    |   movel(p[0.457444, -0.052609, -0.000100, 0.000000, -3.141593, 0.000000],accel_mss,speed_ms,0,0.000)
    |   movel(p[0.456698, -0.052972, -0.000100, 0.000000, -3.141593, 0.000000],accel_mss,speed_ms,0,0.000)
    |   movel(p[0.455801, -0.053375, -0.000100, 0.000000, -3.141593, 0.000000],accel_mss,speed_ms,0,0.000)
    |   movel(p[0.455556, -0.053469, -0.000100, 0.000000, -3.141593, 0.000000],accel_mss,speed_ms,0,0.000)
    |   movel(p[0.455254, -0.053564, -0.000100, 0.000000, 3.141593, 0.000000],accel_mss,speed_ms,0,0.000)
    |   movel(p[0.454943, -0.053645, -0.000100, 0.000000, -3.141593, 0.000000],accel_mss,speed_ms,0,0.000)
    |   movel(p[0.454676, -0.053699, -0.000100, 0.000000, -3.141593, 0.000000],accel_mss,speed_ms,0,0.000)
    |   movel(p[0.454424, -0.053742, -0.000100, 0.000000, -3.141593, 0.000000],accel_mss,speed_ms,0,0.000)
    |   movel(p[0.454164, -0.053792, -0.000100, 0.000000, -3.141593, 0.000000],accel_mss,speed_ms,0,0.000)
    |   movel(p[0.453931, -0.053841, -0.000100, 0.000000, -3.141593, 0.000000],accel_mss,speed_ms,0,0.000)
    |   movel(p[0.453776, -0.053881, -0.000100, 0.000000, -3.141593, 0.000000],accel_mss,speed_ms,0,0.000)
    |   movel(p[0.453611, -0.053919, -0.000100, 0.000000, 3.141593, 0.000000],accel_mss,speed_ms,0,0.000)
    |   movel(p[0.453619, -0.053815, -0.000100, 0.000000, 3.141593, 0.000000],accel_mss,speed_ms,0,0.000)
    |   movel(p[0.453839, -0.053573, -0.000100, 0.000000, -3.141593, 0.000000],accel_mss,speed_ms,0,0.000)
    |   movel(p[0.453990, -0.053422, -0.000100, 0.000000, -3.141593, 0.000000],accel_mss,speed_ms,0,0.000)
    |   movel(p[0.454143, -0.053294, -0.000100, 0.000000, -3.141593, 0.000000],accel_mss,speed_ms,0,0.000)
    |   movel(p[0.454280, -0.053201, -0.000100, 0.000000, -3.141593, 0.000000],accel_mss,speed_ms,0,0.000)
    |   movel(p[0.454467, -0.053141, -0.000100, 0.000000, -3.141593, 0.000000],accel_mss,speed_ms,0,0.000)
    |   movel(p[0.454831, -0.052851, -0.000100, 0.000000, -3.141593, 0.000000],accel_mss,speed_ms,0,0.000)
    |   movel(p[0.455254, -0.052494, -0.000100, 0.000000, -3.141593, 0.000000],accel_mss,speed_ms,0,0.000)
    |   movel(p[0.455726, -0.052070, -0.000100, 0.000000, -3.141593, 0.000000],accel_mss,speed_ms,0,0.000)
    |   movel(p[0.456326, -0.051518, -0.000100, 0.000000, -3.141593, 0.000000],accel_mss,speed_ms,0,0.000)
    |   movel(p[0.456926, -0.050965, -0.000100, 0.000000, -3.141593, 0.000000],accel_mss,speed_ms,0,0.000)
    |   movel(p[0.456738, -0.050804, -0.000100, 0.000000, -3.141593, 0.000000],accel_mss,speed_ms,0,0.000)
    |   movel(p[0.456551, -0.050642, -0.000100, 0.000000, -3.141593, 0.000000],accel_mss,speed_ms,0,0.000)
    |   movel(p[0.456382, -0.050508, -0.000100, 0.000000, -3.141593, 0.000000],accel_mss,speed_ms,0,0.000)
    |   movel(p[0.456187, -0.050372, -0.000100, 0.000000, -3.141593, 0.000000],accel_mss,speed_ms,0,0.000)
    |   movel(p[0.455994, -0.050254, -0.000100, 0.000000, -3.141593, 0.000000],accel_mss,speed_ms,0,0.000)
    |   movel(p[0.455838, -0.050177, -0.000100, 0.000000, 3.141593, 0.000000],accel_mss,speed_ms,0,0.000)
    |   movel(p[0.455624, -0.049995, -0.000100, 0.000000, 3.141593, 0.000000],accel_mss,speed_ms,0,0.000)
    |   movel(p[0.455507, -0.049685, -0.000100, 0.000000, -3.141593, 0.000000],accel_mss,speed_ms,0,0.000)
    |   movel(p[0.455509, -0.049322, -0.000100, 0.000000, -3.141593, 0.000000],accel_mss,speed_ms,0,0.000)
    |   movel(p[0.455638, -0.048995, -0.000100, 0.000000, -3.141593, 0.000000],accel_mss,speed_ms,0,0.000)
    |   movel(p[0.455763, -0.048888, -0.000100, 0.000000, 3.141593, 0.000000],accel_mss,speed_ms,0,0.000)
    |   movel(p[0.455918, -0.048877, -0.000100, 0.000000, 3.141593, 0.000000],accel_mss,speed_ms,0,0.000)
    |   movel(p[0.456158, -0.048983, -0.000100, 0.000000, -3.141593, 0.000000],accel_mss,speed_ms,0,0.000)
    |   movel(p[0.456626, -0.049278, -0.000100, 0.000000, 3.141593, 0.000000],accel_mss,speed_ms,0,0.000)
    |   movel(p[0.456820, -0.049403, -0.000100, 0.000000, -3.141593, 0.000000],accel_mss,speed_ms,0,0.000)
    |   movel(p[0.457032, -0.049532, -0.000100, 0.000000, -3.141593, 0.000000],accel_mss,speed_ms,0,0.000)
    |   movel(p[0.457229, -0.049648, -0.000100, 0.000000, -3.141593, 0.000000],accel_mss,speed_ms,0,0.000)
    |   movel(p[0.457376, -0.049726, -0.000100, 0.000000, -3.141593, 0.000000],accel_mss,speed_ms,0,0.000)
    |   movel(p[0.457509, -0.049798, -0.000100, 0.000000, -3.141593, 0.000000],accel_mss,speed_ms,0,0.000)
    |   movel(p[0.457663, -0.049888, -0.000100, 0.000000, -3.141593, 0.000000],accel_mss,speed_ms,0,0.000)
    |   movel(p[0.457813, -0.049981, -0.000100, 0.000000, -3.141593, 0.000000],accel_mss,speed_ms,0,0.000)
    |   movel(p[0.457933, -0.050062, -0.000100, 0.000000, 3.141593, 0.000000],accel_mss,speed_ms,0,0.000)
    |   movel(p[0.458085, -0.050138, -0.000100, 0.000000, 3.141593, 0.000000],accel_mss,speed_ms,0,0.000)
    |   movel(p[0.458220, -0.050138, -0.000100, 0.000000, -3.141593, 0.000000],accel_mss,speed_ms,0,0.000)
    |   movel(p[0.458374, -0.050057, -0.000100, 0.000000, -3.141593, 0.000000],accel_mss,speed_ms,0,0.000)
    |   movel(p[0.458608, -0.049856, -0.000100, 0.000000, -3.141593, 0.000000],accel_mss,speed_ms,0,0.000)
    |   movel(p[0.458781, -0.049703, -0.000100, 0.000000, -3.141593, 0.000000],accel_mss,speed_ms,0,0.000)
    |   movel(p[0.458954, -0.049564, -0.000100, 0.000000, -3.141593, 0.000000],accel_mss,speed_ms,0,0.000)
    |   movel(p[0.459108, -0.049455, -0.000100, 0.000000, -3.141593, 0.000000],accel_mss,speed_ms,0,0.000)
    |   movel(p[0.459201, -0.049410, -0.000100, 0.000000, -3.141593, 0.000000],accel_mss,speed_ms,0,0.000)
    |   movel(p[0.459315, -0.049350, -0.000100, 0.000000, -3.141593, 0.000000],accel_mss,speed_ms,0,0.000)
    |   movel(p[0.459714, -0.049032, -0.000100, 0.000000, 3.141593, 0.000000],accel_mss,speed_ms,0,0.000)
    |   movel(p[0.460181, -0.048647, -0.000100, 0.000000, -3.141593, 0.000000],accel_mss,speed_ms,0,0.000)
    |   movel(p[0.460701, -0.048201, -0.000100, 0.000000, -3.141593, 0.000000],accel_mss,speed_ms,0,0.000)
    |   movel(p[0.462085, -0.046990, -0.000100, 0.000000, -3.141593, 0.000000],accel_mss,speed_ms,0,0.001)
    |   movel(p[0.462714, -0.046416, -0.000100, 0.000000, -3.141593, 0.000000],accel_mss,speed_ms,0,0.000)
    |   movel(p[0.463064, -0.046063, -0.000100, 0.000000, -3.141593, 0.000000],accel_mss,speed_ms,0,0.000)
    |   movel(p[0.463140, -0.045885, -0.000100, 0.000000, -3.141593, 0.000000],accel_mss,speed_ms,0,0.000)
    |   movel(p[0.463215, -0.045710, -0.000100, 0.000000, -3.141593, 0.000000],accel_mss,speed_ms,0,0.000)
    |   movel(p[0.463291, -0.045611, -0.000100, 0.000000, 3.141593, 0.000000],accel_mss,speed_ms,0,0.000)
    |   movel(p[0.463379, -0.045526, -0.000100, 0.000000, -3.141593, 0.000000],accel_mss,speed_ms,0,0.000)
    |   movel(p[0.463505, -0.045328, -0.000100, 0.000000, -3.141593, 0.000000],accel_mss,speed_ms,0,0.000)
    |   movel(p[0.463516, -0.045062, -0.000100, 0.000000, -3.141593, 0.000000],accel_mss,speed_ms,0,0.000)
    |   movel(p[0.463406, -0.044754, -0.000100, 0.000000, -3.141593, 0.000000],accel_mss,speed_ms,0,0.000)
    |   movel(p[0.463185, -0.044441, -0.000100, 0.000000, -3.141593, 0.000000],accel_mss,speed_ms,0,0.000)
    |   movel(p[0.462587, -0.044166, -0.000100, 0.000000, -3.141593, 0.000000],accel_mss,speed_ms,0,0.000)
    |   movel(p[0.461450, -0.044260, -0.000100, 0.000000, -3.141593, 0.000000],accel_mss,speed_ms,0,0.000)
    |   movel(p[0.460266, -0.044596, -0.000100, 0.000000, -3.141593, 0.000000],accel_mss,speed_ms,0,0.000)
    |   movel(p[0.459446, -0.045117, -0.000100, 0.000000, -3.141593, 0.000000],accel_mss,speed_ms,0,0.000)
    |   movel(p[0.459259, -0.045315, -0.000100, 0.000000, 3.141593, 0.000000],accel_mss,speed_ms,0,0.000)
    |   movel(p[0.459093, -0.045532, -0.000100, 0.000000, -3.141593, 0.000000],accel_mss,speed_ms,0,0.000)
    |   movel(p[0.458970, -0.045736, -0.000100, 0.000000, -3.141593, 0.000000],accel_mss,speed_ms,0,0.000)
    |   movel(p[0.458921, -0.045889, -0.000100, 0.000000, -3.141593, 0.000000],accel_mss,speed_ms,0,0.000)
    |   movel(p[0.458835, -0.046155, -0.000100, 0.000000, -3.141593, 0.000000],accel_mss,speed_ms,0,0.000)
    |   movel(p[0.458710, -0.046179, -0.000100, 0.000000, -3.141593, 0.000000],accel_mss,speed_ms,0,0.000)
    |   movel(p[0.458578, -0.045966, -0.000100, 0.000000, -3.141593, 0.000000],accel_mss,speed_ms,0,0.000)
    |   movel(p[0.458501, -0.045529, -0.000100, 0.000000, -3.141593, 0.000000],accel_mss,speed_ms,0,0.000)
    |   movel(p[0.458463, -0.045191, -0.000100, 0.000000, 3.141593, 0.000000],accel_mss,speed_ms,0,0.000)
    |   movel(p[0.458426, -0.044854, -0.000100, 0.000000, -3.141593, 0.000000],accel_mss,speed_ms,0,0.000)
    |   movel(p[0.457956, -0.044809, -0.000100, 0.000000, -3.141593, 0.000000],accel_mss,speed_ms,0,0.000)
    |   movel(p[0.457486, -0.044764, -0.000100, 0.000000, -3.141593, 0.000000],accel_mss,speed_ms,0,0.000)
    |   movel(p[0.457118, -0.044722, -0.000100, 0.000000, -3.141593, 0.000000],accel_mss,speed_ms,0,0.000)
    |   movel(p[0.456793, -0.044671, -0.000100, 0.000000, -3.141593, 0.000000],accel_mss,speed_ms,0,0.000)
    |   movel(p[0.456525, -0.044617, -0.000100, 0.000000, -3.141593, 0.000000],accel_mss,speed_ms,0,0.000)
    |   movel(p[0.456394, -0.044568, -0.000100, 0.000000, -3.141593, 0.000000],accel_mss,speed_ms,0,0.000)
    |   movel(p[0.456241, -0.044747, -0.000100, 0.000000, -3.141593, 0.000000],accel_mss,speed_ms,0,0.000)
    |   movel(p[0.456164, -0.044906, -0.000100, 0.000000, -3.141593, 0.000000],accel_mss,speed_ms,0,0.000)
    |   movel(p[0.456062, -0.045092, -0.000100, 0.000000, -3.141593, 0.000000],accel_mss,speed_ms,0,0.000)
    |   movel(p[0.455929, -0.045243, -0.000100, 0.000000, 3.141593, 0.000000],accel_mss,speed_ms,0,0.000)
    |   movel(p[0.455772, -0.045351, -0.000100, 0.000000, -3.141593, 0.000000],accel_mss,speed_ms,0,0.000)
    |   movel(p[0.455599, -0.045411, -0.000100, 0.000000, -3.141593, 0.000000],accel_mss,speed_ms,0,0.000)
    |   movel(p[0.455393, -0.045435, -0.000100, 0.000000, -3.141593, 0.000000],accel_mss,speed_ms,0,0.000)
    |   movel(p[0.455279, -0.045400, -0.000100, 0.000000, -3.141593, 0.000000],accel_mss,speed_ms,0,0.000)
    |   movel(p[0.455211, -0.045303, -0.000100, 0.000000, -3.141593, 0.000000],accel_mss,speed_ms,0,0.000)
    |   movel(p[0.455171, -0.045103, -0.000100, 0.000000, -3.141593, 0.000000],accel_mss,speed_ms,0,0.000)
    |   movel(p[0.454942, -0.044704, -0.000100, 0.000000, -3.141593, 0.000000],accel_mss,speed_ms,0,0.000)
    |   movel(p[0.454225, -0.044245, -0.000100, 0.000000, -3.141593, 0.000000],accel_mss,speed_ms,0,0.000)
    |   movel(p[0.453175, -0.043770, -0.000100, 0.000000, -3.141593, 0.000000],accel_mss,speed_ms,0,0.000)
    |   movel(p[0.451809, -0.043308, -0.000100, 0.000000, -3.141593, 0.000000],accel_mss,speed_ms,0,0.001)
    |   movel(p[0.450322, -0.042878, -0.000100, 0.000000, 3.141593, 0.000000],accel_mss,speed_ms,0,0.001)
    |   movel(p[0.449341, -0.042643, -0.000100, 0.000000, -3.141593, 0.000000],accel_mss,speed_ms,0,0.000)
    |   movel(p[0.448468, -0.042508, -0.000100, 0.000000, -3.141593, 0.000000],accel_mss,speed_ms,0,0.000)
    |   movel(p[0.447398, -0.042420, -0.000100, 0.000000, -3.141593, 0.000000],accel_mss,speed_ms,0,0.000)
    |   movel(p[0.445629, -0.042470, -0.000100, 0.000000, -3.141593, 0.000000],accel_mss,speed_ms,0,0.001)
    |   movel(p[0.444085, -0.042832, -0.000100, 0.000000, -3.141593, 0.000000],accel_mss,speed_ms,0,0.001)
    |   movel(p[0.442690, -0.043537, -0.000100, 0.000000, -3.141593, 0.000000],accel_mss,speed_ms,0,0.001)
    |   movel(p[0.441363, -0.044610, -0.000100, 0.000000, -3.141593, 0.000000],accel_mss,speed_ms,0,0.001)
    |   movel(p[0.440975, -0.045000, -0.000100, 0.000000, -3.141593, 0.000000],accel_mss,speed_ms,0,0.000)
    |   movel(p[0.440648, -0.045357, -0.000100, 0.000000, -3.141593, 0.000000],accel_mss,speed_ms,0,0.000)
    |   movel(p[0.440388, -0.045663, -0.000100, 0.000000, -3.141593, 0.000000],accel_mss,speed_ms,0,0.000)
    |   movel(p[0.440351, -0.045769, -0.000100, 0.000000, -3.141593, 0.000000],accel_mss,speed_ms,0,0.000)
    |   movel(p[0.440286, -0.045945, -0.000100, 0.000000, 3.141593, 0.000000],accel_mss,speed_ms,0,0.000)
    |   movel(p[0.440214, -0.046043, -0.000100, 0.000000, -3.141593, 0.000000],accel_mss,speed_ms,0,0.000)
    |   movel(p[0.440129, -0.046126, -0.000100, 0.000000, -3.141593, 0.000000],accel_mss,speed_ms,0,0.000)
    |   movel(p[0.439825, -0.046492, -0.000100, 0.000000, -3.141593, 0.000000],accel_mss,speed_ms,0,0.000)
    |   movel(p[0.439490, -0.047169, -0.000100, 0.000000, -3.141593, 0.000000],accel_mss,speed_ms,0,0.000)
    |   movel(p[0.439225, -0.047864, -0.000100, 0.000000, -3.141593, 0.000000],accel_mss,speed_ms,0,0.000)
    |   movel(p[0.439223, -0.048220, -0.000100, 0.000000, -3.141593, 0.000000],accel_mss,speed_ms,0,0.000)
    |   movel(p[0.439220, -0.048445, -0.000100, 0.000000, -3.141593, 0.000000],accel_mss,speed_ms,0,0.000)
    |   movel(p[0.439086, -0.048517, -0.000100, 0.000000, -3.141593, 0.000000],accel_mss,speed_ms,0,0.000)
    |   movel(p[0.438794, -0.048368, -0.000100, 0.000000, -3.141593, 0.000000],accel_mss,speed_ms,0,0.000)
    |   movel(p[0.438401, -0.048004, -0.000100, 0.000000, -3.141593, 0.000000],accel_mss,speed_ms,0,0.000)
    |   movel(p[0.438193, -0.047803, -0.000100, 0.000000, -3.141593, 0.000000],accel_mss,speed_ms,0,0.000)
    |   movel(p[0.437991, -0.047633, -0.000100, 0.000000, -3.141593, 0.000000],accel_mss,speed_ms,0,0.000)
    |   movel(p[0.437816, -0.047507, -0.000100, 0.000000, 3.141593, 0.000000],accel_mss,speed_ms,0,0.000)
    |   movel(p[0.437634, -0.047455, -0.000100, 0.000000, -3.141593, 0.000000],accel_mss,speed_ms,0,0.000)
    |   movel(p[0.437496, -0.047365, -0.000100, 0.000000, 3.141593, 0.000000],accel_mss,speed_ms,0,0.000)
    |   movel(p[0.437341, -0.047239, -0.000100, 0.000000, -3.141593, 0.000000],accel_mss,speed_ms,0,0.000)
    |   movel(p[0.437189, -0.047090, -0.000100, 0.000000, -3.141593, 0.000000],accel_mss,speed_ms,0,0.000)
    |   movel(p[0.436313, -0.046354, -0.000100, 0.000000, -3.141593, 0.000000],accel_mss,speed_ms,0,0.000)
    |   movel(p[0.434998, -0.045590, -0.000100, 0.000000, 3.141593, 0.000000],accel_mss,speed_ms,0,0.001)
    |   movel(p[0.433551, -0.044941, -0.000100, 0.000000, -3.141593, 0.000000],accel_mss,speed_ms,0,0.001)
    |   movel(p[0.432241, -0.044552, -0.000100, 0.000000, -3.141593, 0.000000],accel_mss,speed_ms,0,0.001)
    |   movel(p[0.431305, -0.044404, -0.000100, 0.000000, -3.141593, 0.000000],accel_mss,speed_ms,0,0.000)
    |   movel(p[0.430304, -0.044342, -0.000100, 0.000000, -3.141593, 0.000000],accel_mss,speed_ms,0,0.000)
    |   movel(p[0.429265, -0.044365, -0.000100, 0.000000, 3.141593, 0.000000],accel_mss,speed_ms,0,0.000)
    |   movel(p[0.428220, -0.044473, -0.000100, 0.000000, -3.141593, 0.000000],accel_mss,speed_ms,0,0.000)
    |   movel(p[0.427528, -0.044623, -0.000100, 0.000000, 3.141593, 0.000000],accel_mss,speed_ms,0,0.000)
    |   movel(p[0.426799, -0.044878, -0.000100, 0.000000, -3.141593, 0.000000],accel_mss,speed_ms,0,0.000)
    |   movel(p[0.426044, -0.045234, -0.000100, 0.000000, -3.141593, 0.000000],accel_mss,speed_ms,0,0.000)
    |   movel(p[0.425276, -0.045686, -0.000100, 0.000000, -3.141593, 0.000000],accel_mss,speed_ms,0,0.000)
    |   movel(p[0.425087, -0.045804, -0.000100, 0.000000, -3.141593, 0.000000],accel_mss,speed_ms,0,0.000)
    |   movel(p[0.424892, -0.045920, -0.000100, 0.000000, 3.141593, 0.000000],accel_mss,speed_ms,0,0.000)
    |   movel(p[0.424717, -0.046019, -0.000100, 0.000000, 3.141593, 0.000000],accel_mss,speed_ms,0,0.000)
    |   movel(p[0.424601, -0.046077, -0.000100, 0.000000, -3.141593, 0.000000],accel_mss,speed_ms,0,0.000)
    |   movel(p[0.424480, -0.046142, -0.000100, 0.000000, -3.141593, 0.000000],accel_mss,speed_ms,0,0.000)
    |   movel(p[0.424281, -0.046274, -0.000100, 0.000000, -3.141593, 0.000000],accel_mss,speed_ms,0,0.000)
    |   movel(p[0.424055, -0.046434, -0.000100, 0.000000, 3.141593, 0.000000],accel_mss,speed_ms,0,0.000)
    |   movel(p[0.423829, -0.046604, -0.000100, 0.000000, -3.141593, 0.000000],accel_mss,speed_ms,0,0.000)
    |   movel(p[0.423610, -0.046767, -0.000100, 0.000000, -3.141593, 0.000000],accel_mss,speed_ms,0,0.000)
    |   movel(p[0.423402, -0.046904, -0.000100, 0.000000, 3.141593, 0.000000],accel_mss,speed_ms,0,0.000)
    |   movel(p[0.423225, -0.047008, -0.000100, 0.000000, 3.141593, 0.000000],accel_mss,speed_ms,0,0.000)
    |   movel(p[0.422935, -0.047109, -0.000100, 0.000000, -3.141593, 0.000000],accel_mss,speed_ms,0,0.000)
    |   movel(p[0.422672, -0.047388, -0.000100, 0.000000, 3.141593, 0.000000],accel_mss,speed_ms,0,0.000)
    |   movel(p[0.422465, -0.047699, -0.000100, 0.000000, -3.141593, 0.000000],accel_mss,speed_ms,0,0.000)
    |   movel(p[0.422470, -0.047879, -0.000100, 0.000000, -3.141593, 0.000000],accel_mss,speed_ms,0,0.000)
    |   movel(p[0.422558, -0.047959, -0.000100, 0.000000, -3.141593, 0.000000],accel_mss,speed_ms,0,0.000)
    |   movel(p[0.422809, -0.048074, -0.000100, 0.000000, 3.141593, 0.000000],accel_mss,speed_ms,0,0.000)
    |   movel(p[0.423123, -0.048195, -0.000100, 0.000000, -3.141593, 0.000000],accel_mss,speed_ms,0,0.000)
    |   movel(p[0.423476, -0.048306, -0.000100, 0.000000, 3.141593, 0.000000],accel_mss,speed_ms,0,0.000)
    |   movel(p[0.423831, -0.048414, -0.000100, 0.000000, -3.141593, 0.000000],accel_mss,speed_ms,0,0.000)
    |   movel(p[0.424153, -0.048526, -0.000100, 0.000000, -3.141593, 0.000000],accel_mss,speed_ms,0,0.000)
    |   movel(p[0.424417, -0.048630, -0.000100, 0.000000, -3.141593, 0.000000],accel_mss,speed_ms,0,0.000)
    |   movel(p[0.424518, -0.048696, -0.000100, 0.000000, -3.141593, 0.000000],accel_mss,speed_ms,0,0.000)
    |   movel(p[0.424691, -0.048790, -0.000100, 0.000000, -3.141593, 0.000000],accel_mss,speed_ms,0,0.000)
    |   movel(p[0.424803, -0.048819, -0.000100, 0.000000, -3.141593, 0.000000],accel_mss,speed_ms,0,0.000)
    |   movel(p[0.424908, -0.048829, -0.000100, 0.000000, -3.141593, 0.000000],accel_mss,speed_ms,0,0.000)
    |   movel(p[0.425036, -0.048845, -0.000100, 0.000000, -3.141593, 0.000000],accel_mss,speed_ms,0,0.000)
    |   movel(p[0.425230, -0.048903, -0.000100, 0.000000, 3.141593, 0.000000],accel_mss,speed_ms,0,0.000)
    |   movel(p[0.425448, -0.048984, -0.000100, 0.000000, -3.141593, 0.000000],accel_mss,speed_ms,0,0.000)
    |   movel(p[0.425659, -0.049081, -0.000100, 0.000000, -3.141593, 0.000000],accel_mss,speed_ms,0,0.000)
    |   movel(p[0.425911, -0.049179, -0.000100, 0.000000, -3.141593, 0.000000],accel_mss,speed_ms,0,0.000)
    |   movel(p[0.426235, -0.049257, -0.000100, 0.000000, -3.141593, 0.000000],accel_mss,speed_ms,0,0.000)
    |   movel(p[0.426586, -0.049306, -0.000100, 0.000000, -3.141593, 0.000000],accel_mss,speed_ms,0,0.000)
    |   movel(p[0.426920, -0.049319, -0.000100, 0.000000, -3.141593, 0.000000],accel_mss,speed_ms,0,0.000)
    |   movel(p[0.427388, -0.049310, -0.000100, 0.000000, -3.141593, 0.000000],accel_mss,speed_ms,0,0.000)
    |   movel(p[0.428446, -0.049289, -0.000100, 0.000000, 3.141593, 0.000000],accel_mss,speed_ms,0,0.000)
    |   movel(p[0.429706, -0.049264, -0.000100, 0.000000, -3.141593, 0.000000],accel_mss,speed_ms,0,0.001)
    |   movel(p[0.431055, -0.049237, -0.000100, 0.000000, -3.141593, 0.000000],accel_mss,speed_ms,0,0.001)
    |   movel(p[0.433370, -0.049228, -0.000100, 0.000000, -3.141593, 0.000000],accel_mss,speed_ms,0,0.001)
    |   movel(p[0.435193, -0.049311, -0.000100, 0.000000, -3.141593, 0.000000],accel_mss,speed_ms,0,0.001)
    |   movel(p[0.436687, -0.049489, -0.000100, 0.000000, -3.141593, 0.000000],accel_mss,speed_ms,0,0.001)
    |   movel(p[0.437970, -0.049777, -0.000100, 0.000000, -3.141593, 0.000000],accel_mss,speed_ms,0,0.001)
    |   movel(p[0.438501, -0.049999, -0.000100, 0.000000, -3.141593, 0.000000],accel_mss,speed_ms,0,0.000)
    |   movel(p[0.438479, -0.050152, -0.000100, 0.000000, -3.141593, 0.000000],accel_mss,speed_ms,0,0.000)
    |   movel(p[0.437782, -0.050237, -0.000100, 0.000000, -3.141593, 0.000000],accel_mss,speed_ms,0,0.000)
    |   movel(p[0.435923, -0.050249, -0.000100, 0.000000, 3.141593, 0.000000],accel_mss,speed_ms,0,0.001)
    |   movel(p[0.433512, -0.050292, -0.000100, 0.000000, 3.141593, 0.000000],accel_mss,speed_ms,0,0.001)
    |   movel(p[0.431714, -0.050442, -0.000100, 0.000000, -3.141593, 0.000000],accel_mss,speed_ms,0,0.001)
    |   movel(p[0.430039, -0.050745, -0.000100, 0.000000, -3.141593, 0.000000],accel_mss,speed_ms,0,0.001)
    |   movel(p[0.428051, -0.051269, -0.000100, 0.000000, -3.141593, 0.000000],accel_mss,speed_ms,0,0.001)
    |   movel(p[0.427120, -0.051615, -0.000100, 0.000000, -3.141593, 0.000000],accel_mss,speed_ms,0,0.000)
    |   movel(p[0.425780, -0.052258, -0.000100, 0.000000, -3.141593, 0.000000],accel_mss,speed_ms,0,0.001)
    |   movel(p[0.424487, -0.052945, -0.000100, 0.000000, -3.141593, 0.000000],accel_mss,speed_ms,0,0.001)
    |   movel(p[0.423864, -0.053391, -0.000100, 0.000000, -3.141593, 0.000000],accel_mss,speed_ms,0,0.000)
    |   movel(p[0.423754, -0.053482, -0.000100, 0.000000, -3.141593, 0.000000],accel_mss,speed_ms,0,0.000)
    |   movel(p[0.423639, -0.053559, -0.000100, 0.000000, -3.141593, 0.000000],accel_mss,speed_ms,0,0.000)
    |   movel(p[0.423535, -0.053614, -0.000100, 0.000000, -3.141593, 0.000000],accel_mss,speed_ms,0,0.000)
    |   movel(p[0.423234, -0.053725, -0.000100, 0.000000, -3.141593, 0.000000],accel_mss,speed_ms,0,0.000)
    |   movel(p[0.421486, -0.055471, -0.000100, 0.000000, -3.141593, 0.000000],accel_mss,speed_ms,0,0.001)
    |   movel(p[0.419747, -0.057225, -0.000100, 0.000000, -3.141593, 0.000000],accel_mss,speed_ms,0,0.001)
    |   movel(p[0.419651, -0.057459, -0.000100, 0.000000, -3.141593, 0.000000],accel_mss,speed_ms,0,0.000)
    |   movel(p[0.419474, -0.057743, -0.000100, 0.000000, 3.141593, 0.000000],accel_mss,speed_ms,0,0.000)
    |   movel(p[0.419280, -0.057968, -0.000100, 0.000000, -3.141593, 0.000000],accel_mss,speed_ms,0,0.000)
    |   movel(p[0.419051, -0.058204, -0.000100, 0.000000, -3.141593, 0.000000],accel_mss,speed_ms,0,0.000)
    |   movel(p[0.418821, -0.058440, -0.000100, 0.000000, -3.141593, 0.000000],accel_mss,speed_ms,0,0.000)
    |   movel(p[0.418627, -0.058665, -0.000100, 0.000000, 3.141593, 0.000000],accel_mss,speed_ms,0,0.000)
    |   movel(p[0.418480, -0.058860, -0.000100, 0.000000, -3.141593, 0.000000],accel_mss,speed_ms,0,0.000)
    |   movel(p[0.418418, -0.059049, -0.000100, 0.000000, -3.141593, 0.000000],accel_mss,speed_ms,0,0.000)
    |   movel(p[0.418230, -0.059284, -0.000100, 0.000000, -3.141593, 0.000000],accel_mss,speed_ms,0,0.000)
    |   movel(p[0.417988, -0.059559, -0.000100, 0.000000, -3.141593, 0.000000],accel_mss,speed_ms,0,0.000)
    |   movel(p[0.417701, -0.059854, -0.000100, 0.000000, -3.141593, 0.000000],accel_mss,speed_ms,0,0.000)
    |   movel(p[0.417413, -0.060146, -0.000100, 0.000000, -3.141593, 0.000000],accel_mss,speed_ms,0,0.000)
    |   movel(p[0.417171, -0.060410, -0.000100, 0.000000, -3.141593, 0.000000],accel_mss,speed_ms,0,0.000)
    |   movel(p[0.416977, -0.060638, -0.000100, 0.000000, -3.141593, 0.000000],accel_mss,speed_ms,0,0.000)
    |   movel(p[0.416978, -0.060756, -0.000100, 0.000000, -3.141593, 0.000000],accel_mss,speed_ms,0,0.000)
    |   movel(p[0.417072, -0.060794, -0.000100, 0.000000, -3.141593, 0.000000],accel_mss,speed_ms,0,0.000)
    |   movel(p[0.417205, -0.060821, -0.000100, 0.000000, 3.141593, 0.000000],accel_mss,speed_ms,0,0.000)
    |   movel(p[0.417363, -0.060830, -0.000100, 0.000000, -3.141593, 0.000000],accel_mss,speed_ms,0,0.000)
    |   movel(p[0.417987, -0.060788, -0.000100, 0.000000, -3.141593, 0.000000],accel_mss,speed_ms,0,0.000)
    |   movel(p[0.419857, -0.060521, -0.000100, 0.000000, -3.141593, 0.000000],accel_mss,speed_ms,0,0.001)
    |   movel(p[0.421692, -0.060242, -0.000100, 0.000000, -3.141593, 0.000000],accel_mss,speed_ms,0,0.001)
    |   movel(p[0.422501, -0.060076, -0.000100, 0.000000, -3.141593, 0.000000],accel_mss,speed_ms,0,0.000)
    |   movel(p[0.422801, -0.060010, -0.000100, 0.000000, -3.141593, 0.000000],accel_mss,speed_ms,0,0.000)
    |   movel(p[0.423353, -0.059908, -0.000100, 0.000000, -3.141593, 0.000000],accel_mss,speed_ms,0,0.000)
    |   movel(p[0.423999, -0.059798, -0.000100, 0.000000, -3.141593, 0.000000],accel_mss,speed_ms,0,0.000)
    |   movel(p[0.424665, -0.059692, -0.000100, 0.000000, -3.141593, 0.000000],accel_mss,speed_ms,0,0.000)
    |   movel(p[0.426937, -0.059271, -0.000100, 0.000000, 3.141593, 0.000000],accel_mss,speed_ms,0,0.001)
    |   movel(p[0.429210, -0.058707, -0.000100, 0.000000, -3.141593, 0.000000],accel_mss,speed_ms,0,0.001)
    |   movel(p[0.431205, -0.058082, -0.000100, 0.000000, -3.141593, 0.000000],accel_mss,speed_ms,0,0.001)
    |   movel(p[0.432551, -0.057484, -0.000100, 0.000000, -3.141593, 0.000000],accel_mss,speed_ms,0,0.001)
    |   movel(p[0.432888, -0.057299, -0.000100, 0.000000, -3.141593, 0.000000],accel_mss,speed_ms,0,0.000)
    |   movel(p[0.433221, -0.057117, -0.000100, 0.000000, -3.141593, 0.000000],accel_mss,speed_ms,0,0.000)
    |   movel(p[0.433509, -0.056959, -0.000100, 0.000000, -3.141593, 0.000000],accel_mss,speed_ms,0,0.000)
    |   movel(p[0.433676, -0.056868, -0.000100, 0.000000, -3.141593, 0.000000],accel_mss,speed_ms,0,0.000)
    |   movel(p[0.434155, -0.056529, -0.000100, 0.000000, 3.141593, 0.000000],accel_mss,speed_ms,0,0.000)
    |   movel(p[0.434933, -0.055797, -0.000100, 0.000000, -3.141593, 0.000000],accel_mss,speed_ms,0,0.000)
    |   movel(p[0.435685, -0.055018, -0.000100, 0.000000, -3.141593, 0.000000],accel_mss,speed_ms,0,0.000)
    |   movel(p[0.436125, -0.054454, -0.000100, 0.000000, -3.141593, 0.000000],accel_mss,speed_ms,0,0.000)
    |   movel(p[0.436484, -0.053902, -0.000100, 0.000000, -3.141593, 0.000000],accel_mss,speed_ms,0,0.000)
    |   movel(p[0.436721, -0.053523, -0.000100, 0.000000, -3.141593, 0.000000],accel_mss,speed_ms,0,0.000)
    |   movel(p[0.436891, -0.053227, -0.000100, 0.000000, -3.141593, 0.000000],accel_mss,speed_ms,0,0.000)
    |   movel(p[0.437030, -0.052954, -0.000100, 0.000000, -3.141593, 0.000000],accel_mss,speed_ms,0,0.000)
    |   movel(p[0.437118, -0.052806, -0.000100, 0.000000, -3.141593, 0.000000],accel_mss,speed_ms,0,0.000)
    |   movel(p[0.437281, -0.052597, -0.000100, 0.000000, -3.141593, 0.000000],accel_mss,speed_ms,0,0.000)
    |   movel(p[0.437480, -0.052371, -0.000100, 0.000000, -3.141593, 0.000000],accel_mss,speed_ms,0,0.000)
    |   movel(p[0.437687, -0.052160, -0.000100, 0.000000, 3.141593, 0.000000],accel_mss,speed_ms,0,0.000)
    |   movel(p[0.438114, -0.051835, -0.000100, 0.000000, -3.141593, 0.000000],accel_mss,speed_ms,0,0.000)
    |   movel(p[0.438368, -0.051872, -0.000100, 0.000000, -3.141593, 0.000000],accel_mss,speed_ms,0,0.000)
    |   movel(p[0.438519, -0.052214, -0.000100, 0.000000, -3.141593, 0.000000],accel_mss,speed_ms,0,0.000)
    |   movel(p[0.438570, -0.053117, -0.000100, 0.000000, -3.141593, 0.000000],accel_mss,speed_ms,0,0.000)
    |   movel(p[0.438471, -0.054698, -0.000100, 0.000000, -3.141593, 0.000000],accel_mss,speed_ms,0,0.001)
    |   movel(p[0.438094, -0.056047, -0.000100, 0.000000, -3.141593, 0.000000],accel_mss,speed_ms,0,0.001)
    |   movel(p[0.437375, -0.057323, -0.000100, 0.000000, -3.141593, 0.000000],accel_mss,speed_ms,0,0.001)
    |   movel(p[0.436235, -0.058691, -0.000100, 0.000000, -3.141593, 0.000000],accel_mss,speed_ms,0,0.001)
    |   movel(p[0.435936, -0.058993, -0.000100, 0.000000, -3.141593, 0.000000],accel_mss,speed_ms,0,0.000)
    |   movel(p[0.435657, -0.059248, -0.000100, 0.000000, -3.141593, 0.000000],accel_mss,speed_ms,0,0.000)
    |   movel(p[0.435418, -0.059445, -0.000100, 0.000000, -3.141593, 0.000000],accel_mss,speed_ms,0,0.000)
    |   movel(p[0.435319, -0.059479, -0.000100, 0.000000, 3.141593, 0.000000],accel_mss,speed_ms,0,0.000)
    |   movel(p[0.435101, -0.059587, -0.000100, 0.000000, -3.141593, 0.000000],accel_mss,speed_ms,0,0.000)
    |   movel(p[0.434953, -0.059705, -0.000100, 0.000000, -3.141593, 0.000000],accel_mss,speed_ms,0,0.000)
    |   movel(p[0.434809, -0.059845, -0.000100, 0.000000, -3.141593, 0.000000],accel_mss,speed_ms,0,0.000)
    |   movel(p[0.434643, -0.060003, -0.000100, 0.000000, -3.141593, 0.000000],accel_mss,speed_ms,0,0.000)
    |   movel(p[0.434428, -0.060174, -0.000100, 0.000000, -3.141593, 0.000000],accel_mss,speed_ms,0,0.000)
    |   movel(p[0.434200, -0.060332, -0.000100, 0.000000, -3.141593, 0.000000],accel_mss,speed_ms,0,0.000)
    |   movel(p[0.433995, -0.060450, -0.000100, 0.000000, -3.141593, 0.000000],accel_mss,speed_ms,0,0.000)
    |   movel(p[0.433799, -0.060550, -0.000100, 0.000000, -3.141593, 0.000000],accel_mss,speed_ms,0,0.000)
    |   movel(p[0.433597, -0.060657, -0.000100, 0.000000, -3.141593, 0.000000],accel_mss,speed_ms,0,0.000)
    |   movel(p[0.433418, -0.060754, -0.000100, 0.000000, -3.141593, 0.000000],accel_mss,speed_ms,0,0.000)
    |   movel(p[0.433301, -0.060821, -0.000100, 0.000000, -3.141593, 0.000000],accel_mss,speed_ms,0,0.000)
    |   movel(p[0.432770, -0.061109, -0.000100, 0.000000, 3.141593, 0.000000],accel_mss,speed_ms,0,0.000)
    |   movel(p[0.432187, -0.061374, -0.000100, 0.000000, -3.141593, 0.000000],accel_mss,speed_ms,0,0.000)
    |   movel(p[0.431648, -0.061577, -0.000100, 0.000000, -3.141593, 0.000000],accel_mss,speed_ms,0,0.000)
    |   movel(p[0.431280, -0.061659, -0.000100, 0.000000, -3.141593, 0.000000],accel_mss,speed_ms,0,0.000)
    |   movel(p[0.431044, -0.061693, -0.000100, 0.000000, -3.141593, 0.000000],accel_mss,speed_ms,0,0.000)
    |   movel(p[0.430689, -0.061762, -0.000100, 0.000000, -3.141593, 0.000000],accel_mss,speed_ms,0,0.000)
    |   movel(p[0.430291, -0.061847, -0.000100, 0.000000, 3.141593, 0.000000],accel_mss,speed_ms,0,0.000)
    |   movel(p[0.429906, -0.061938, -0.000100, 0.000000, -3.141593, 0.000000],accel_mss,speed_ms,0,0.000)
    |   movel(p[0.427696, -0.062362, -0.000100, 0.000000, -3.141593, 0.000000],accel_mss,speed_ms,0,0.001)
    |   movel(p[0.425276, -0.062585, -0.000100, 0.000000, -3.141593, 0.000000],accel_mss,speed_ms,0,0.001)
    |   movel(p[0.422775, -0.062602, -0.000100, 0.000000, 3.141593, 0.000000],accel_mss,speed_ms,0,blend_radius_m)
    |   movel(p[0.420320, -0.062405, -0.000100, 0.000000, -3.141593, 0.000000],accel_mss,speed_ms,0,0.001)
    |   movel(p[0.419535, -0.062319, -0.000100, 0.000000, -3.141593, 0.000000],accel_mss,speed_ms,0,0.000)
    |   movel(p[0.418658, -0.062247, -0.000100, 0.000000, -3.141593, 0.000000],accel_mss,speed_ms,0,0.000)
    |   movel(p[0.417824, -0.062196, -0.000100, 0.000000, -3.141593, 0.000000],accel_mss,speed_ms,0,0.000)
    |   movel(p[0.417182, -0.062180, -0.000100, 0.000000, -3.141593, 0.000000],accel_mss,speed_ms,0,0.000)
    |   movel(p[0.416306, -0.062191, -0.000100, 0.000000, -3.141593, 0.000000],accel_mss,speed_ms,0,0.000)
    |   movel(p[0.415937, -0.062247, -0.000100, 0.000000, -3.141593, 0.000000],accel_mss,speed_ms,0,0.000)
    |   movel(p[0.415660, -0.062389, -0.000100, 0.000000, -3.141593, 0.000000],accel_mss,speed_ms,0,0.000)
    |   movel(p[0.415283, -0.062721, -0.000100, 0.000000, -3.141593, 0.000000],accel_mss,speed_ms,0,0.000)
    |   movel(p[0.415059, -0.062922, -0.000100, 0.000000, -3.141593, 0.000000],accel_mss,speed_ms,0,0.000)
    |   movel(p[0.414843, -0.063075, -0.000100, 0.000000, -3.141593, 0.000000],accel_mss,speed_ms,0,0.000)
    |   movel(p[0.414662, -0.063170, -0.000100, 0.000000, -3.141593, 0.000000],accel_mss,speed_ms,0,0.000)
    |   movel(p[0.414426, -0.062902, -0.000100, 0.000000, -3.141593, 0.000000],accel_mss,speed_ms,0,0.000)
    |   movel(p[0.414484, -0.061805, -0.000100, 0.000000, -3.141593, 0.000000],accel_mss,speed_ms,0,0.000)
    |   movel(p[0.414620, -0.060625, -0.000100, 0.000000, -3.141593, 0.000000],accel_mss,speed_ms,0,0.000)
    |   movel(p[0.414838, -0.059587, -0.000100, 0.000000, -3.141593, 0.000000],accel_mss,speed_ms,0,0.000)
    |   movel(p[0.415173, -0.058419, -0.000100, 0.000000, 3.141593, 0.000000],accel_mss,speed_ms,0,0.000)
    |   movel(p[0.415458, -0.057633, -0.000100, 0.000000, -3.141593, 0.000000],accel_mss,speed_ms,0,0.000)
    |   movel(p[0.415812, -0.056906, -0.000100, 0.000000, -3.141593, 0.000000],accel_mss,speed_ms,0,0.000)
    |   movel(p[0.416371, -0.055954, -0.000100, 0.000000, 3.141593, 0.000000],accel_mss,speed_ms,0,0.000)
    |   movel(p[0.416484, -0.055765, -0.000100, 0.000000, -3.141593, 0.000000],accel_mss,speed_ms,0,0.000)
    |   movel(p[0.416595, -0.055570, -0.000100, 0.000000, -3.141593, 0.000000],accel_mss,speed_ms,0,0.000)
    |   movel(p[0.416690, -0.055395, -0.000100, 0.000000, -3.141593, 0.000000],accel_mss,speed_ms,0,0.000)
    |   movel(p[0.416745, -0.055279, -0.000100, 0.000000, -3.141593, 0.000000],accel_mss,speed_ms,0,0.000)
    |   movel(p[0.416971, -0.054932, -0.000100, 0.000000, 3.141593, 0.000000],accel_mss,speed_ms,0,0.000)
    |   movel(p[0.417623, -0.054250, -0.000100, 0.000000, -3.141593, 0.000000],accel_mss,speed_ms,0,0.000)
    |   movel(p[0.418321, -0.053565, -0.000100, 0.000000, -3.141593, 0.000000],accel_mss,speed_ms,0,0.000)
    |   movel(p[0.418535, -0.053479, -0.000100, 0.000000, -3.141593, 0.000000],accel_mss,speed_ms,0,0.000)
    |   movel(p[0.418734, -0.053391, -0.000100, 0.000000, -3.141593, 0.000000],accel_mss,speed_ms,0,0.000)
    |   movel(p[0.418859, -0.053294, -0.000100, 0.000000, -3.141593, 0.000000],accel_mss,speed_ms,0,0.000)
    |   movel(p[0.418976, -0.053179, -0.000100, 0.000000, -3.141593, 0.000000],accel_mss,speed_ms,0,0.000)
    |   movel(p[0.419093, -0.053064, -0.000100, 0.000000, -3.141593, 0.000000],accel_mss,speed_ms,0,0.000)
    |   movel(p[0.419220, -0.052967, -0.000100, 0.000000, 3.141593, 0.000000],accel_mss,speed_ms,0,0.000)
    |   movel(p[0.419339, -0.052899, -0.000100, 0.000000, 3.141593, 0.000000],accel_mss,speed_ms,0,0.000)
    |   movel(p[0.419512, -0.052859, -0.000100, 0.000000, -3.141593, 0.000000],accel_mss,speed_ms,0,0.000)
    |   movel(p[0.419629, -0.052794, -0.000100, 0.000000, 3.141593, 0.000000],accel_mss,speed_ms,0,0.000)
    |   movel(p[0.419753, -0.052700, -0.000100, 0.000000, -3.141593, 0.000000],accel_mss,speed_ms,0,0.000)
    |   movel(p[0.419866, -0.052590, -0.000100, 0.000000, -3.141593, 0.000000],accel_mss,speed_ms,0,0.000)
    |   movel(p[0.420000, -0.052461, -0.000100, 0.000000, -3.141593, 0.000000],accel_mss,speed_ms,0,0.000)
    |   movel(p[0.420190, -0.052314, -0.000100, 0.000000, 3.141593, 0.000000],accel_mss,speed_ms,0,0.000)
    |   movel(p[0.420401, -0.052171, -0.000100, 0.000000, -3.141593, 0.000000],accel_mss,speed_ms,0,0.000)
    |   movel(p[0.420602, -0.052056, -0.000100, 0.000000, -3.141593, 0.000000],accel_mss,speed_ms,0,0.000)
    |   movel(p[0.421674, -0.051491, -0.000100, 0.000000, -3.141593, 0.000000],accel_mss,speed_ms,0,0.000)
    |   movel(p[0.422593, -0.050977, -0.000100, 0.000000, -3.141593, 0.000000],accel_mss,speed_ms,0,0.000)
    |   movel(p[0.423373, -0.050520, -0.000100, 0.000000, -3.141593, 0.000000],accel_mss,speed_ms,0,0.000)
    |   movel(p[0.423452, -0.050405, -0.000100, 0.000000, -3.141593, 0.000000],accel_mss,speed_ms,0,0.000)
    |   movel(p[0.423286, -0.050100, -0.000100, 0.000000, -3.141593, 0.000000],accel_mss,speed_ms,0,0.000)
    |   movel(p[0.422190, -0.049694, -0.000100, 0.000000, 3.141593, 0.000000],accel_mss,speed_ms,0,0.000)
    |   movel(p[0.420757, -0.049299, -0.000100, 0.000000, -3.141593, 0.000000],accel_mss,speed_ms,0,0.001)
    |   movel(p[0.419077, -0.048975, -0.000100, 0.000000, -3.141593, 0.000000],accel_mss,speed_ms,0,0.001)
    |   movel(p[0.418599, -0.048885, -0.000100, 0.000000, -3.141593, 0.000000],accel_mss,speed_ms,0,0.000)
    |   movel(p[0.418240, -0.048786, -0.000100, 0.000000, -3.141593, 0.000000],accel_mss,speed_ms,0,0.000)
    |   movel(p[0.417991, -0.048681, -0.000100, 0.000000, -3.141593, 0.000000],accel_mss,speed_ms,0,0.000)
    |   movel(p[0.417893, -0.048574, -0.000100, 0.000000, -3.141593, 0.000000],accel_mss,speed_ms,0,0.000)
    |   movel(p[0.417884, -0.048443, -0.000100, 0.000000, -3.141593, 0.000000],accel_mss,speed_ms,0,0.000)
    |   movel(p[0.417952, -0.048195, -0.000100, 0.000000, -3.141593, 0.000000],accel_mss,speed_ms,0,0.000)
    |   movel(p[0.418064, -0.047903, -0.000100, 0.000000, -3.141593, 0.000000],accel_mss,speed_ms,0,0.000)
    |   movel(p[0.418213, -0.047599, -0.000100, 0.000000, 3.141593, 0.000000],accel_mss,speed_ms,0,0.000)
    |   movel(p[0.418363, -0.047305, -0.000100, 0.000000, -3.141593, 0.000000],accel_mss,speed_ms,0,0.000)
    |   movel(p[0.418477, -0.047045, -0.000100, 0.000000, -3.141593, 0.000000],accel_mss,speed_ms,0,0.000)
    |   movel(p[0.418556, -0.046831, -0.000100, 0.000000, -3.141593, 0.000000],accel_mss,speed_ms,0,0.000)
    |   movel(p[0.418397, -0.046726, -0.000100, 0.000000, 3.141593, 0.000000],accel_mss,speed_ms,0,0.000)
    |   movel(p[0.418193, -0.046808, -0.000100, 0.000000, -3.141593, 0.000000],accel_mss,speed_ms,0,0.000)
    |   movel(p[0.417988, -0.046985, -0.000100, 0.000000, -3.141593, 0.000000],accel_mss,speed_ms,0,0.000)
    |   movel(p[0.417842, -0.047213, -0.000100, 0.000000, -3.141593, 0.000000],accel_mss,speed_ms,0,0.000)
    |   movel(p[0.417655, -0.047597, -0.000100, 0.000000, -3.141593, 0.000000],accel_mss,speed_ms,0,0.000)
    |   movel(p[0.417457, -0.047946, -0.000100, 0.000000, -3.141593, 0.000000],accel_mss,speed_ms,0,0.000)
    |   movel(p[0.417253, -0.048251, -0.000100, 0.000000, -3.141593, 0.000000],accel_mss,speed_ms,0,0.000)
    |   movel(p[0.417050, -0.048502, -0.000100, 0.000000, 3.141593, 0.000000],accel_mss,speed_ms,0,0.000)
    |   movel(p[0.416954, -0.048617, -0.000100, 0.000000, 3.141593, 0.000000],accel_mss,speed_ms,0,0.000)
    |   movel(p[0.416874, -0.048733, -0.000100, 0.000000, -3.141593, 0.000000],accel_mss,speed_ms,0,0.000)
    |   movel(p[0.416816, -0.048837, -0.000100, 0.000000, -3.141593, 0.000000],accel_mss,speed_ms,0,0.000)
    |   movel(p[0.416782, -0.048975, -0.000100, 0.000000, -3.141593, 0.000000],accel_mss,speed_ms,0,0.000)
    |   movel(p[0.416690, -0.049134, -0.000100, 0.000000, -3.141593, 0.000000],accel_mss,speed_ms,0,0.000)
    |   movel(p[0.416569, -0.049320, -0.000100, 0.000000, 3.141593, 0.000000],accel_mss,speed_ms,0,0.000)
    |   movel(p[0.416426, -0.049517, -0.000100, 0.000000, -3.141593, 0.000000],accel_mss,speed_ms,0,0.000)
    |   movel(p[0.416282, -0.049716, -0.000100, 0.000000, -3.141593, 0.000000],accel_mss,speed_ms,0,0.000)
    |   movel(p[0.416161, -0.049906, -0.000100, 0.000000, -3.141593, 0.000000],accel_mss,speed_ms,0,0.000)
    |   movel(p[0.416070, -0.050069, -0.000100, 0.000000, -3.141593, 0.000000],accel_mss,speed_ms,0,0.000)
    |   movel(p[0.416036, -0.050217, -0.000100, 0.000000, -3.141593, 0.000000],accel_mss,speed_ms,0,0.000)
    |   movel(p[0.415921, -0.050389, -0.000100, 0.000000, -3.141593, 0.000000],accel_mss,speed_ms,0,0.000)
    |   movel(p[0.415840, -0.050467, -0.000100, 0.000000, -3.141593, 0.000000],accel_mss,speed_ms,0,0.000)
    |   movel(p[0.415753, -0.050561, -0.000100, 0.000000, -3.141593, 0.000000],accel_mss,speed_ms,0,0.000)
    |   movel(p[0.415663, -0.050704, -0.000100, 0.000000, -3.141593, 0.000000],accel_mss,speed_ms,0,0.000)
    |   movel(p[0.415585, -0.050869, -0.000100, 0.000000, -3.141593, 0.000000],accel_mss,speed_ms,0,0.000)
    |   movel(p[0.415532, -0.051031, -0.000100, 0.000000, -3.141593, 0.000000],accel_mss,speed_ms,0,0.000)
    |   movel(p[0.415469, -0.051214, -0.000100, 0.000000, -3.141593, 0.000000],accel_mss,speed_ms,0,0.000)
    |   movel(p[0.415356, -0.051447, -0.000100, 0.000000, -3.141593, 0.000000],accel_mss,speed_ms,0,0.000)
    |   movel(p[0.415215, -0.051688, -0.000100, 0.000000, -3.141593, 0.000000],accel_mss,speed_ms,0,0.000)
    |   movel(p[0.415068, -0.051901, -0.000100, 0.000000, 3.141593, 0.000000],accel_mss,speed_ms,0,0.000)
    |   movel(p[0.414927, -0.052092, -0.000100, 0.000000, -3.141593, 0.000000],accel_mss,speed_ms,0,0.000)
    |   movel(p[0.414808, -0.052269, -0.000100, 0.000000, 3.141593, 0.000000],accel_mss,speed_ms,0,0.000)
    |   movel(p[0.414717, -0.052419, -0.000100, 0.000000, -3.141593, 0.000000],accel_mss,speed_ms,0,0.000)
    |   movel(p[0.414686, -0.052547, -0.000100, 0.000000, -3.141593, 0.000000],accel_mss,speed_ms,0,0.000)
    |   movel(p[0.414499, -0.052976, -0.000100, 0.000000, -3.141593, 0.000000],accel_mss,speed_ms,0,0.000)
    |   movel(p[0.414277, -0.053470, -0.000100, 0.000000, -3.141593, 0.000000],accel_mss,speed_ms,0,0.000)
    |   movel(p[0.414014, -0.054039, -0.000100, 0.000000, -3.141593, 0.000000],accel_mss,speed_ms,0,0.000)
    |   movel(p[0.413741, -0.054625, -0.000100, 0.000000, -3.141593, 0.000000],accel_mss,speed_ms,0,0.000)
    |   movel(p[0.413488, -0.055173, -0.000100, 0.000000, -3.141593, 0.000000],accel_mss,speed_ms,0,0.000)
    |   movel(p[0.413278, -0.055634, -0.000100, 0.000000, -3.141593, 0.000000],accel_mss,speed_ms,0,0.000)
    |   movel(p[0.413189, -0.055841, -0.000100, 0.000000, -3.141593, 0.000000],accel_mss,speed_ms,0,0.000)
    |   movel(p[0.413125, -0.055995, -0.000100, 0.000000, 3.141593, 0.000000],accel_mss,speed_ms,0,0.000)
    |   movel(p[0.413048, -0.056179, -0.000100, 0.000000, -3.141593, 0.000000],accel_mss,speed_ms,0,0.000)
    |   movel(p[0.412970, -0.056363, -0.000100, 0.000000, -3.141593, 0.000000],accel_mss,speed_ms,0,0.000)
    |   movel(p[0.412904, -0.056516, -0.000100, 0.000000, 3.141593, 0.000000],accel_mss,speed_ms,0,0.000)
    |   movel(p[0.412828, -0.056701, -0.000100, 0.000000, -3.141593, 0.000000],accel_mss,speed_ms,0,0.000)
    |   movel(p[0.412709, -0.057008, -0.000100, 0.000000, -3.141593, 0.000000],accel_mss,speed_ms,0,0.000)
    |   movel(p[0.412575, -0.057361, -0.000100, 0.000000, 3.141593, 0.000000],accel_mss,speed_ms,0,0.000)
    |   movel(p[0.412444, -0.057716, -0.000100, 0.000000, -3.141593, 0.000000],accel_mss,speed_ms,0,0.000)
    |   movel(p[0.412315, -0.058047, -0.000100, 0.000000, -3.141593, 0.000000],accel_mss,speed_ms,0,0.000)
    |   movel(p[0.412188, -0.058326, -0.000100, 0.000000, -3.141593, 0.000000],accel_mss,speed_ms,0,0.000)
    |   movel(p[0.412073, -0.058545, -0.000100, 0.000000, 3.141593, 0.000000],accel_mss,speed_ms,0,0.000)
    |   movel(p[0.411961, -0.058558, -0.000100, 0.000000, 3.141593, 0.000000],accel_mss,speed_ms,0,0.000)
    |   movel(p[0.411886, -0.058480, -0.000100, 0.000000, -3.141593, 0.000000],accel_mss,speed_ms,0,0.000)
    |   movel(p[0.411807, -0.058371, -0.000100, 0.000000, -3.141593, 0.000000],accel_mss,speed_ms,0,0.000)
    |   movel(p[0.411735, -0.058241, -0.000100, 0.000000, -3.141593, 0.000000],accel_mss,speed_ms,0,0.000)
    |   movel(p[0.411427, -0.057586, -0.000100, 0.000000, -3.141593, 0.000000],accel_mss,speed_ms,0,0.000)
    |   movel(p[0.411100, -0.056821, -0.000100, 0.000000, -3.141593, 0.000000],accel_mss,speed_ms,0,0.000)
    |   movel(p[0.410799, -0.056062, -0.000100, 0.000000, -3.141593, 0.000000],accel_mss,speed_ms,0,0.000)
    |   movel(p[0.410576, -0.055429, -0.000100, 0.000000, -3.141593, 0.000000],accel_mss,speed_ms,0,0.000)
    |   movel(p[0.410458, -0.055091, -0.000100, 0.000000, 3.141593, 0.000000],accel_mss,speed_ms,0,0.000)
    |   movel(p[0.410327, -0.054759, -0.000100, 0.000000, -3.141593, 0.000000],accel_mss,speed_ms,0,0.000)
    |   movel(p[0.410200, -0.054475, -0.000100, 0.000000, -3.141593, 0.000000],accel_mss,speed_ms,0,0.000)
    |   movel(p[0.410104, -0.054308, -0.000100, 0.000000, -3.141593, 0.000000],accel_mss,speed_ms,0,0.000)
    |   movel(p[0.410026, -0.054177, -0.000100, 0.000000, -3.141593, 0.000000],accel_mss,speed_ms,0,0.000)
    |   movel(p[0.409960, -0.054027, -0.000100, 0.000000, -3.141593, 0.000000],accel_mss,speed_ms,0,0.000)
    |   movel(p[0.409915, -0.053881, -0.000100, 0.000000, 3.141593, 0.000000],accel_mss,speed_ms,0,0.000)
    |   movel(p[0.409901, -0.053766, -0.000100, 0.000000, -3.141593, 0.000000],accel_mss,speed_ms,0,0.000)
    |   movel(p[0.409878, -0.053607, -0.000100, 0.000000, -3.141593, 0.000000],accel_mss,speed_ms,0,0.000)
    |   movel(p[0.409746, -0.053178, -0.000100, 0.000000, -3.141593, 0.000000],accel_mss,speed_ms,0,0.000)
    |   movel(p[0.409576, -0.052669, -0.000100, 0.000000, -3.141593, 0.000000],accel_mss,speed_ms,0,0.000)
    |   movel(p[0.409374, -0.052112, -0.000100, 0.000000, -3.141593, 0.000000],accel_mss,speed_ms,0,0.000)
    |   movel(p[0.409167, -0.051540, -0.000100, 0.000000, 3.141593, 0.000000],accel_mss,speed_ms,0,0.000)
    |   movel(p[0.408978, -0.050985, -0.000100, 0.000000, 3.141593, 0.000000],accel_mss,speed_ms,0,0.000)
    |   movel(p[0.408829, -0.050510, -0.000100, 0.000000, 3.141593, 0.000000],accel_mss,speed_ms,0,0.000)
    |   movel(p[0.408767, -0.050254, -0.000100, 0.000000, -3.141593, 0.000000],accel_mss,speed_ms,0,0.000)
    |   movel(p[0.408713, -0.050007, -0.000100, 0.000000, -3.141593, 0.000000],accel_mss,speed_ms,0,0.000)
    |   movel(p[0.408601, -0.049589, -0.000100, 0.000000, 3.141593, 0.000000],accel_mss,speed_ms,0,0.000)
    |   movel(p[0.408463, -0.049107, -0.000100, 0.000000, -3.141593, 0.000000],accel_mss,speed_ms,0,0.000)
    |   movel(p[0.408315, -0.048622, -0.000100, 0.000000, 3.141593, 0.000000],accel_mss,speed_ms,0,0.000)
    |   movel(p[0.408061, -0.047778, -0.000100, 0.000000, -3.141593, 0.000000],accel_mss,speed_ms,0,0.000)
    |   movel(p[0.407844, -0.046980, -0.000100, 0.000000, -3.141593, 0.000000],accel_mss,speed_ms,0,0.000)
    |   movel(p[0.407677, -0.046281, -0.000100, 0.000000, -3.141593, 0.000000],accel_mss,speed_ms,0,0.000)
    |   movel(p[0.407581, -0.045754, -0.000100, 0.000000, -3.141593, 0.000000],accel_mss,speed_ms,0,0.000)
    |   movel(p[0.407550, -0.045561, -0.000100, 0.000000, -3.141593, 0.000000],accel_mss,speed_ms,0,0.000)
    |   movel(p[0.407458, -0.045072, -0.000100, 0.000000, -3.141593, 0.000000],accel_mss,speed_ms,0,0.000)
    |   movel(p[0.407347, -0.044488, -0.000100, 0.000000, 3.141593, 0.000000],accel_mss,speed_ms,0,0.000)
    |   movel(p[0.407223, -0.043852, -0.000100, 0.000000, -3.141593, 0.000000],accel_mss,speed_ms,0,0.000)
    |   movel(p[0.406642, -0.040112, -0.000100, 0.000000, -3.141593, 0.000000],accel_mss,speed_ms,0,blend_radius_m)
    |   movel(p[0.406475, -0.036856, -0.000100, 0.000000, -3.141593, 0.000000],accel_mss,speed_ms,0,blend_radius_m)
    |   movel(p[0.406714, -0.033998, -0.000100, 0.000000, 3.141593, 0.000000],accel_mss,speed_ms,0,blend_radius_m)
    |   movel(p[0.407363, -0.031466, -0.000100, 0.000000, -3.141593, 0.000000],accel_mss,speed_ms,0,blend_radius_m)
    |   movel(p[0.407465, -0.031164, -0.000100, 0.000000, -3.141593, 0.000000],accel_mss,speed_ms,0,0.000)
    |   movel(p[0.407539, -0.030910, -0.000100, 0.000000, -3.141593, 0.000000],accel_mss,speed_ms,0,0.000)
    |   movel(p[0.407586, -0.030707, -0.000100, 0.000000, -3.141593, 0.000000],accel_mss,speed_ms,0,0.000)
    |   movel(p[0.407588, -0.030558, -0.000100, 0.000000, -3.141593, 0.000000],accel_mss,speed_ms,0,0.000)
    |   movel(p[0.407661, -0.030425, -0.000100, 0.000000, -3.141593, 0.000000],accel_mss,speed_ms,0,0.000)
    |   movel(p[0.407763, -0.030266, -0.000100, 0.000000, -3.141593, 0.000000],accel_mss,speed_ms,0,0.000)
    |   movel(p[0.407901, -0.030048, -0.000100, 0.000000, -3.141593, 0.000000],accel_mss,speed_ms,0,0.000)
    |   movel(p[0.408089, -0.029713, -0.000100, 0.000000, 3.141593, 0.000000],accel_mss,speed_ms,0,0.000)
    |   movel(p[0.408290, -0.029332, -0.000100, 0.000000, 3.141593, 0.000000],accel_mss,speed_ms,0,0.000)
    |   movel(p[0.408475, -0.028960, -0.000100, 0.000000, 3.141593, 0.000000],accel_mss,speed_ms,0,0.000)
    |   movel(p[0.408777, -0.028436, -0.000100, 0.000000, -3.141593, 0.000000],accel_mss,speed_ms,0,0.000)
    |   movel(p[0.409207, -0.027865, -0.000100, 0.000000, 3.141593, 0.000000],accel_mss,speed_ms,0,0.000)
    |   movel(p[0.409821, -0.027172, -0.000100, 0.000000, -3.141593, 0.000000],accel_mss,speed_ms,0,0.000)
    |   movel(p[0.410715, -0.026256, -0.000100, 0.000000, 3.141593, 0.000000],accel_mss,speed_ms,0,0.001)
    |   movel(p[0.411791, -0.025199, -0.000100, 0.000000, -3.141593, 0.000000],accel_mss,speed_ms,0,0.001)
    |   movel(p[0.412378, -0.024692, -0.000100, 0.000000, -3.141593, 0.000000],accel_mss,speed_ms,0,0.000)
    |   movel(p[0.412856, -0.024394, -0.000100, 0.000000, -3.141593, 0.000000],accel_mss,speed_ms,0,0.000)
    |   movel(p[0.413419, -0.024170, -0.000100, 0.000000, -3.141593, 0.000000],accel_mss,speed_ms,0,0.000)
    |   movel(p[0.414219, -0.023977, -0.000100, 0.000000, 3.141593, 0.000000],accel_mss,speed_ms,0,0.000)
    |   movel(p[0.414969, -0.023908, -0.000100, 0.000000, -3.141593, 0.000000],accel_mss,speed_ms,0,0.000)
    |   movel(p[0.415712, -0.023961, -0.000100, 0.000000, -3.141593, 0.000000],accel_mss,speed_ms,0,0.000)
    |   movel(p[0.416493, -0.024138, -0.000100, 0.000000, -3.141593, 0.000000],accel_mss,speed_ms,0,0.000)
    |   movel(p[0.417152, -0.024402, -0.000100, 0.000000, -3.141593, 0.000000],accel_mss,speed_ms,0,0.000)
    |   movel(p[0.417689, -0.024765, -0.000100, 0.000000, -3.141593, 0.000000],accel_mss,speed_ms,0,0.000)
    |   movel(p[0.418126, -0.025251, -0.000100, 0.000000, -3.141593, 0.000000],accel_mss,speed_ms,0,0.000)
    |   movel(p[0.418491, -0.025879, -0.000100, 0.000000, 3.141593, 0.000000],accel_mss,speed_ms,0,0.000)
    |   movel(p[0.418688, -0.026345, -0.000100, 0.000000, -3.141593, 0.000000],accel_mss,speed_ms,0,0.000)
    |   movel(p[0.418832, -0.026792, -0.000100, 0.000000, -3.141593, 0.000000],accel_mss,speed_ms,0,0.000)
    |   movel(p[0.418914, -0.027157, -0.000100, 0.000000, 3.141593, 0.000000],accel_mss,speed_ms,0,0.000)
    |   movel(p[0.418815, -0.027221, -0.000100, 0.000000, 3.141593, 0.000000],accel_mss,speed_ms,0,0.000)
    |   movel(p[0.418676, -0.027160, -0.000100, 0.000000, -3.141593, 0.000000],accel_mss,speed_ms,0,0.000)
    |   movel(p[0.418512, -0.027085, -0.000100, 0.000000, -3.141593, 0.000000],accel_mss,speed_ms,0,0.000)
    |   movel(p[0.418328, -0.026995, -0.000100, 0.000000, -3.141593, 0.000000],accel_mss,speed_ms,0,0.000)
    |   movel(p[0.417708, -0.026785, -0.000100, 0.000000, 3.141593, 0.000000],accel_mss,speed_ms,0,0.000)
    |   movel(p[0.416784, -0.026652, -0.000100, 0.000000, -3.141593, 0.000000],accel_mss,speed_ms,0,0.000)
    |   movel(p[0.415844, -0.026610, -0.000100, 0.000000, -3.141593, 0.000000],accel_mss,speed_ms,0,0.000)
    |   movel(p[0.415160, -0.026697, -0.000100, 0.000000, -3.141593, 0.000000],accel_mss,speed_ms,0,0.000)
    |   movel(p[0.414493, -0.026982, -0.000100, 0.000000, -3.141593, 0.000000],accel_mss,speed_ms,0,0.000)
    |   movel(p[0.413903, -0.027469, -0.000100, 0.000000, -3.141593, 0.000000],accel_mss,speed_ms,0,0.000)
    |   movel(p[0.413454, -0.028103, -0.000100, 0.000000, -3.141593, 0.000000],accel_mss,speed_ms,0,0.000)
    |   movel(p[0.413198, -0.028816, -0.000100, 0.000000, 3.141593, 0.000000],accel_mss,speed_ms,0,0.000)
    |   movel(p[0.413065, -0.030052, -0.000100, 0.000000, -3.141593, 0.000000],accel_mss,speed_ms,0,0.000)
    |   movel(p[0.413157, -0.031395, -0.000100, 0.000000, -3.141593, 0.000000],accel_mss,speed_ms,0,0.001)
    |   movel(p[0.413456, -0.032723, -0.000100, 0.000000, -3.141593, 0.000000],accel_mss,speed_ms,0,0.001)
    |   movel(p[0.413943, -0.033914, -0.000100, 0.000000, -3.141593, 0.000000],accel_mss,speed_ms,0,0.001)
    |   movel(p[0.414352, -0.034638, -0.000100, 0.000000, -3.141593, 0.000000],accel_mss,speed_ms,0,0.000)
    |   movel(p[0.414695, -0.035075, -0.000100, 0.000000, -3.141593, 0.000000],accel_mss,speed_ms,0,0.000)
    |   movel(p[0.415109, -0.035401, -0.000100, 0.000000, 3.141593, 0.000000],accel_mss,speed_ms,0,0.000)
    |   movel(p[0.415746, -0.035742, -0.000100, 0.000000, -3.141593, 0.000000],accel_mss,speed_ms,0,0.000)
    |   movel(p[0.416704, -0.036059, -0.000100, 0.000000, -3.141593, 0.000000],accel_mss,speed_ms,0,0.000)
    |   movel(p[0.417784, -0.036165, -0.000100, 0.000000, -3.141593, 0.000000],accel_mss,speed_ms,0,0.000)
    |   movel(p[0.418858, -0.036058, -0.000100, 0.000000, -3.141593, 0.000000],accel_mss,speed_ms,0,0.000)
    |   movel(p[0.419801, -0.035741, -0.000100, 0.000000, -3.141593, 0.000000],accel_mss,speed_ms,0,0.000)
    |   movel(p[0.421163, -0.034799, -0.000100, 0.000000, -3.141593, 0.000000],accel_mss,speed_ms,0,0.001)
    |   movel(p[0.422404, -0.033354, -0.000100, 0.000000, -3.141593, 0.000000],accel_mss,speed_ms,0,0.001)
    |   movel(p[0.423439, -0.031525, -0.000100, 0.000000, -3.141593, 0.000000],accel_mss,speed_ms,0,0.001)
    |   movel(p[0.424184, -0.029437, -0.000100, 0.000000, -3.141593, 0.000000],accel_mss,speed_ms,0,0.001)
    |   movel(p[0.424417, -0.028220, -0.000100, 0.000000, -3.141593, 0.000000],accel_mss,speed_ms,0,0.000)
    |   movel(p[0.424522, -0.026759, -0.000100, 0.000000, 3.141593, 0.000000],accel_mss,speed_ms,0,0.001)
    |   movel(p[0.424498, -0.025374, -0.000100, 0.000000, -3.141593, 0.000000],accel_mss,speed_ms,0,0.001)
    |   movel(p[0.424316, -0.024454, -0.000100, 0.000000, -3.141593, 0.000000],accel_mss,speed_ms,0,0.000)
    |   movel(p[0.423542, -0.022676, -0.000100, 0.000000, -3.141593, 0.000000],accel_mss,speed_ms,0,0.001)
    |   movel(p[0.422552, -0.021230, -0.000100, 0.000000, 3.141593, 0.000000],accel_mss,speed_ms,0,0.001)
    |   movel(p[0.421294, -0.020061, -0.000100, 0.000000, -3.141593, 0.000000],accel_mss,speed_ms,0,0.001)
    |   movel(p[0.419726, -0.019110, -0.000100, 0.000000, -3.141593, 0.000000],accel_mss,speed_ms,0,0.001)
    |   movel(p[0.419051, -0.018782, -0.000100, 0.000000, 3.141593, 0.000000],accel_mss,speed_ms,0,0.000)
    |   movel(p[0.418376, -0.018454, -0.000100, 0.000000, 3.141593, 0.000000],accel_mss,speed_ms,0,0.000)
    |   movel(p[0.417251, -0.018457, -0.000100, 0.000000, -3.141593, 0.000000],accel_mss,speed_ms,0,0.000)
    |   movel(p[0.416126, -0.018459, -0.000100, 0.000000, 3.141593, 0.000000],accel_mss,speed_ms,0,0.000)
    |   movel(p[0.414975, -0.018475, -0.000100, 0.000000, -3.141593, 0.000000],accel_mss,speed_ms,0,0.000)
    |   movel(p[0.414162, -0.018521, -0.000100, 0.000000, 3.141593, 0.000000],accel_mss,speed_ms,0,0.000)
    |   movel(p[0.413531, -0.018604, -0.000100, 0.000000, -3.141593, 0.000000],accel_mss,speed_ms,0,0.000)
    |   movel(p[0.412976, -0.018736, -0.000100, 0.000000, -3.141593, 0.000000],accel_mss,speed_ms,0,0.000)
    |   movel(p[0.412149, -0.019018, -0.000100, 0.000000, -3.141593, 0.000000],accel_mss,speed_ms,0,0.000)
    |   movel(p[0.411337, -0.019362, -0.000100, 0.000000, -3.141593, 0.000000],accel_mss,speed_ms,0,0.000)
    |   movel(p[0.410653, -0.019706, -0.000100, 0.000000, 3.141593, 0.000000],accel_mss,speed_ms,0,0.000)
    |   movel(p[0.410348, -0.019958, -0.000100, 0.000000, -3.141593, 0.000000],accel_mss,speed_ms,0,0.000)
    |   movel(p[0.410265, -0.020042, -0.000100, 0.000000, 3.141593, 0.000000],accel_mss,speed_ms,0,0.000)
    |   movel(p[0.410169, -0.020114, -0.000100, 0.000000, 3.141593, 0.000000],accel_mss,speed_ms,0,0.000)
    |   movel(p[0.410075, -0.020163, -0.000100, 0.000000, -3.141593, 0.000000],accel_mss,speed_ms,0,0.000)
    |   movel(p[0.409751, -0.020279, -0.000100, 0.000000, -3.141593, 0.000000],accel_mss,speed_ms,0,0.000)
    |   movel(p[0.408744, -0.021264, -0.000100, 0.000000, -3.141593, 0.000000],accel_mss,speed_ms,0,0.001)
    |   movel(p[0.407750, -0.022265, -0.000100, 0.000000, -3.141593, 0.000000],accel_mss,speed_ms,0,0.001)
    |   movel(p[0.407651, -0.022510, -0.000100, 0.000000, 3.141593, 0.000000],accel_mss,speed_ms,0,0.000)
    |   movel(p[0.407518, -0.022751, -0.000100, 0.000000, 3.141593, 0.000000],accel_mss,speed_ms,0,0.000)
    |   movel(p[0.407373, -0.022927, -0.000100, 0.000000, -3.141593, 0.000000],accel_mss,speed_ms,0,0.000)
    |   movel(p[0.407201, -0.023104, -0.000100, 0.000000, -3.141593, 0.000000],accel_mss,speed_ms,0,0.000)
    |   movel(p[0.407028, -0.023279, -0.000100, 0.000000, 3.141593, 0.000000],accel_mss,speed_ms,0,0.000)
    |   movel(p[0.406883, -0.023448, -0.000100, 0.000000, -3.141593, 0.000000],accel_mss,speed_ms,0,0.000)
    |   movel(p[0.406774, -0.023594, -0.000100, 0.000000, -3.141593, 0.000000],accel_mss,speed_ms,0,0.000)
    |   movel(p[0.406729, -0.023750, -0.000100, 0.000000, 3.141593, 0.000000],accel_mss,speed_ms,0,0.000)
    |   movel(p[0.406607, -0.023948, -0.000100, 0.000000, -3.141593, 0.000000],accel_mss,speed_ms,0,0.000)
    |   movel(p[0.406450, -0.024179, -0.000100, 0.000000, 3.141593, 0.000000],accel_mss,speed_ms,0,0.000)
    |   movel(p[0.406263, -0.024429, -0.000100, 0.000000, -3.141593, 0.000000],accel_mss,speed_ms,0,0.000)
    |   movel(p[0.405869, -0.024949, -0.000100, 0.000000, -3.141593, 0.000000],accel_mss,speed_ms,0,0.000)
    |   movel(p[0.405604, -0.025336, -0.000100, 0.000000, 3.141593, 0.000000],accel_mss,speed_ms,0,0.000)
    |   movel(p[0.405411, -0.025675, -0.000100, 0.000000, -3.141593, 0.000000],accel_mss,speed_ms,0,0.000)
    |   movel(p[0.405250, -0.026029, -0.000100, 0.000000, -3.141593, 0.000000],accel_mss,speed_ms,0,0.000)
    |   movel(p[0.405180, -0.026194, -0.000100, 0.000000, -3.141593, 0.000000],accel_mss,speed_ms,0,0.000)
    |   movel(p[0.405094, -0.026382, -0.000100, 0.000000, -3.141593, 0.000000],accel_mss,speed_ms,0,0.000)
    |   movel(p[0.405004, -0.026562, -0.000100, 0.000000, -3.141593, 0.000000],accel_mss,speed_ms,0,0.000)
    |   movel(p[0.404927, -0.026704, -0.000100, 0.000000, 3.141593, 0.000000],accel_mss,speed_ms,0,0.000)
    |   movel(p[0.404435, -0.027648, -0.000100, 0.000000, -3.141593, 0.000000],accel_mss,speed_ms,0,0.000)
    |   movel(p[0.404053, -0.028589, -0.000100, 0.000000, -3.141593, 0.000000],accel_mss,speed_ms,0,0.000)
    |   movel(p[0.403686, -0.029778, -0.000100, 0.000000, 3.141593, 0.000000],accel_mss,speed_ms,0,0.000)
    |   movel(p[0.403225, -0.031579, -0.000100, 0.000000, -3.141593, 0.000000],accel_mss,speed_ms,0,0.001)
    |   movel(p[0.402730, -0.034727, -0.000100, 0.000000, -3.141593, 0.000000],accel_mss,speed_ms,0,blend_radius_m)
    |   movel(p[0.402653, -0.035889, -0.000100, 0.000000, -3.141593, 0.000000],accel_mss,speed_ms,0,0.000)
    |   movel(p[0.402593, -0.037053, -0.000100, 0.000000, -3.141593, 0.000000],accel_mss,speed_ms,0,0.000)
    |   movel(p[0.402549, -0.038217, -0.000100, 0.000000, -3.141593, 0.000000],accel_mss,speed_ms,0,0.000)
    |   movel(p[0.402522, -0.039381, -0.000100, 0.000000, -3.141593, 0.000000],accel_mss,speed_ms,0,0.000)
    |   movel(p[0.402510, -0.040597, -0.000100, 0.000000, 3.141593, 0.000000],accel_mss,speed_ms,0,0.000)
    |   movel(p[0.402516, -0.041814, -0.000100, 0.000000, -3.141593, 0.000000],accel_mss,speed_ms,0,0.000)
    |   movel(p[0.402539, -0.043030, -0.000100, 0.000000, -3.141593, 0.000000],accel_mss,speed_ms,0,0.000)
    |   movel(p[0.402579, -0.044246, -0.000100, 0.000000, -3.141593, 0.000000],accel_mss,speed_ms,0,0.000)
    |   movel(p[0.402632, -0.045245, -0.000100, 0.000000, -3.141593, 0.000000],accel_mss,speed_ms,0,0.000)
    |   movel(p[0.402711, -0.046242, -0.000100, 0.000000, -3.141593, 0.000000],accel_mss,speed_ms,0,0.000)
    |   movel(p[0.402815, -0.047237, -0.000100, 0.000000, -3.141593, 0.000000],accel_mss,speed_ms,0,0.000)
    |   movel(p[0.402944, -0.048229, -0.000100, 0.000000, -3.141593, 0.000000],accel_mss,speed_ms,0,0.000)
    |   movel(p[0.403132, -0.049463, -0.000100, 0.000000, -3.141593, 0.000000],accel_mss,speed_ms,0,0.000)
    |   movel(p[0.403335, -0.050634, -0.000100, 0.000000, -3.141593, 0.000000],accel_mss,speed_ms,0,0.000)
    |   movel(p[0.403539, -0.051675, -0.000100, 0.000000, -3.141593, 0.000000],accel_mss,speed_ms,0,0.000)
    |   movel(p[0.403731, -0.052504, -0.000100, 0.000000, -3.141593, 0.000000],accel_mss,speed_ms,0,0.000)
    |   movel(p[0.403796, -0.052771, -0.000100, 0.000000, -3.141593, 0.000000],accel_mss,speed_ms,0,0.000)
    |   movel(p[0.403866, -0.053079, -0.000100, 0.000000, -3.141593, 0.000000],accel_mss,speed_ms,0,0.000)
    |   movel(p[0.403929, -0.053380, -0.000100, 0.000000, -3.141593, 0.000000],accel_mss,speed_ms,0,0.000)
    |   movel(p[0.403975, -0.053621, -0.000100, 0.000000, 3.141593, 0.000000],accel_mss,speed_ms,0,0.000)
    |   movel(p[0.404156, -0.054383, -0.000100, 0.000000, -3.141593, 0.000000],accel_mss,speed_ms,0,0.000)
    |   movel(p[0.404611, -0.055842, -0.000100, 0.000000, -3.141593, 0.000000],accel_mss,speed_ms,0,0.001)
    |   movel(p[0.405096, -0.057291, -0.000100, 0.000000, -3.141593, 0.000000],accel_mss,speed_ms,0,0.001)
    |   movel(p[0.405412, -0.058070, -0.000100, 0.000000, -3.141593, 0.000000],accel_mss,speed_ms,0,0.000)
    |   movel(p[0.405522, -0.058316, -0.000100, 0.000000, 3.141593, 0.000000],accel_mss,speed_ms,0,0.000)
    |   movel(p[0.405616, -0.058544, -0.000100, 0.000000, -3.141593, 0.000000],accel_mss,speed_ms,0,0.000)
    |   movel(p[0.405687, -0.058737, -0.000100, 0.000000, -3.141593, 0.000000],accel_mss,speed_ms,0,0.000)
    |   movel(p[0.405773, -0.059126, -0.000100, 0.000000, -3.141593, 0.000000],accel_mss,speed_ms,0,0.000)
    |   movel(p[0.406661, -0.060906, -0.000100, 0.000000, -3.141593, 0.000000],accel_mss,speed_ms,0,0.001)
    |   movel(p[0.407514, -0.062576, -0.000100, 0.000000, 3.141593, 0.000000],accel_mss,speed_ms,0,0.001)
    |   movel(p[0.407894, -0.063181, -0.000100, 0.000000, -3.141593, 0.000000],accel_mss,speed_ms,0,0.000)
    |   movel(p[0.408030, -0.063375, -0.000100, 0.000000, -3.141593, 0.000000],accel_mss,speed_ms,0,0.000)
    |   movel(p[0.408146, -0.063560, -0.000100, 0.000000, -3.141593, 0.000000],accel_mss,speed_ms,0,0.000)
    |   movel(p[0.408231, -0.063720, -0.000100, 0.000000, -3.141593, 0.000000],accel_mss,speed_ms,0,0.000)
    |   movel(p[0.408266, -0.063868, -0.000100, 0.000000, -3.141593, 0.000000],accel_mss,speed_ms,0,0.000)
    |   movel(p[0.408316, -0.063955, -0.000100, 0.000000, -3.141593, 0.000000],accel_mss,speed_ms,0,0.000)
    |   movel(p[0.408389, -0.064046, -0.000100, 0.000000, -3.141593, 0.000000],accel_mss,speed_ms,0,0.000)
    |   movel(p[0.408474, -0.064128, -0.000100, 0.000000, -3.141593, 0.000000],accel_mss,speed_ms,0,0.000)
    |   movel(p[0.408554, -0.064207, -0.000100, 0.000000, -3.141593, 0.000000],accel_mss,speed_ms,0,0.000)
    |   movel(p[0.408611, -0.064293, -0.000100, 0.000000, -3.141593, 0.000000],accel_mss,speed_ms,0,0.000)
    |   movel(p[0.408626, -0.064429, -0.000100, 0.000000, -3.141593, 0.000000],accel_mss,speed_ms,0,0.000)
    |   movel(p[0.408641, -0.064565, -0.000100, 0.000000, -3.141593, 0.000000],accel_mss,speed_ms,0,0.000)
    |   movel(p[0.408697, -0.064651, -0.000100, 0.000000, 3.141593, 0.000000],accel_mss,speed_ms,0,0.000)
    |   movel(p[0.408777, -0.064730, -0.000100, 0.000000, 3.141593, 0.000000],accel_mss,speed_ms,0,0.000)
    |   movel(p[0.408863, -0.064812, -0.000100, 0.000000, -3.141593, 0.000000],accel_mss,speed_ms,0,0.000)
    |   movel(p[0.408935, -0.064903, -0.000100, 0.000000, -3.141593, 0.000000],accel_mss,speed_ms,0,0.000)
    |   movel(p[0.408985, -0.064990, -0.000100, 0.000000, -3.141593, 0.000000],accel_mss,speed_ms,0,0.000)
    |   movel(p[0.409020, -0.065139, -0.000100, 0.000000, -3.141593, 0.000000],accel_mss,speed_ms,0,0.000)
    |   movel(p[0.409111, -0.065302, -0.000100, 0.000000, -3.141593, 0.000000],accel_mss,speed_ms,0,0.000)
    |   movel(p[0.409232, -0.065492, -0.000100, 0.000000, -3.141593, 0.000000],accel_mss,speed_ms,0,0.000)
    |   movel(p[0.409376, -0.065691, -0.000100, 0.000000, -3.141593, 0.000000],accel_mss,speed_ms,0,0.000)
    |   movel(p[0.409519, -0.065890, -0.000100, 0.000000, 3.141593, 0.000000],accel_mss,speed_ms,0,0.000)
    |   movel(p[0.409640, -0.066082, -0.000100, 0.000000, -3.141593, 0.000000],accel_mss,speed_ms,0,0.000)
    |   movel(p[0.409730, -0.066247, -0.000100, 0.000000, -3.141593, 0.000000],accel_mss,speed_ms,0,0.000)
    |   movel(p[0.409770, -0.066408, -0.000100, 0.000000, 3.141593, 0.000000],accel_mss,speed_ms,0,0.000)
    |   movel(p[0.409839, -0.066518, -0.000100, 0.000000, -3.141593, 0.000000],accel_mss,speed_ms,0,0.000)
    |   movel(p[0.409936, -0.066639, -0.000100, 0.000000, -3.141593, 0.000000],accel_mss,speed_ms,0,0.000)
    |   movel(p[0.410051, -0.066754, -0.000100, 0.000000, -3.141593, 0.000000],accel_mss,speed_ms,0,0.000)
    |   movel(p[0.410165, -0.066867, -0.000100, 0.000000, -3.141593, 0.000000],accel_mss,speed_ms,0,0.000)
    |   movel(p[0.410263, -0.066983, -0.000100, 0.000000, 3.141593, 0.000000],accel_mss,speed_ms,0,0.000)
    |   movel(p[0.410332, -0.067087, -0.000100, 0.000000, -3.141593, 0.000000],accel_mss,speed_ms,0,0.000)
    |   movel(p[0.410372, -0.067235, -0.000100, 0.000000, -3.141593, 0.000000],accel_mss,speed_ms,0,0.000)
    |   movel(p[0.410505, -0.067464, -0.000100, 0.000000, 3.141593, 0.000000],accel_mss,speed_ms,0,0.000)
    |   movel(p[0.410675, -0.067733, -0.000100, 0.000000, -3.141593, 0.000000],accel_mss,speed_ms,0,0.000)
    |   movel(p[0.410876, -0.068029, -0.000100, 0.000000, -3.141593, 0.000000],accel_mss,speed_ms,0,0.000)
    |   movel(p[0.411077, -0.068322, -0.000100, 0.000000, -3.141593, 0.000000],accel_mss,speed_ms,0,0.000)
    |   movel(p[0.411246, -0.068583, -0.000100, 0.000000, -3.141593, 0.000000],accel_mss,speed_ms,0,0.000)
    |   movel(p[0.411384, -0.068806, -0.000100, 0.000000, -3.141593, 0.000000],accel_mss,speed_ms,0,0.000)
    |   movel(p[0.411418, -0.068922, -0.000100, 0.000000, -3.141593, 0.000000],accel_mss,speed_ms,0,0.000)
    |   movel(p[0.411548, -0.069111, -0.000100, 0.000000, -3.141593, 0.000000],accel_mss,speed_ms,0,0.000)
    |   movel(p[0.411710, -0.069333, -0.000100, 0.000000, 3.141593, 0.000000],accel_mss,speed_ms,0,0.000)
    |   movel(p[0.411902, -0.069579, -0.000100, 0.000000, 3.141593, 0.000000],accel_mss,speed_ms,0,0.000)
    |   movel(p[0.412102, -0.069835, -0.000100, 0.000000, -3.141593, 0.000000],accel_mss,speed_ms,0,0.000)
    |   movel(p[0.412286, -0.070086, -0.000100, 0.000000, -3.141593, 0.000000],accel_mss,speed_ms,0,0.000)
    |   movel(p[0.412435, -0.070305, -0.000100, 0.000000, -3.141593, 0.000000],accel_mss,speed_ms,0,0.000)
    |   movel(p[0.412502, -0.070429, -0.000100, 0.000000, -3.141593, 0.000000],accel_mss,speed_ms,0,0.000)
    |   movel(p[0.412570, -0.070555, -0.000100, 0.000000, -3.141593, 0.000000],accel_mss,speed_ms,0,0.000)
    |   movel(p[0.412726, -0.070786, -0.000100, 0.000000, -3.141593, 0.000000],accel_mss,speed_ms,0,0.000)
    |   movel(p[0.412917, -0.071054, -0.000100, 0.000000, -3.141593, 0.000000],accel_mss,speed_ms,0,0.000)
    |   movel(p[0.413126, -0.071329, -0.000100, 0.000000, -3.141593, 0.000000],accel_mss,speed_ms,0,0.000)
    |   movel(p[0.413334, -0.071604, -0.000100, 0.000000, -3.141593, 0.000000],accel_mss,speed_ms,0,0.000)
    |   movel(p[0.413525, -0.071872, -0.000100, 0.000000, -3.141593, 0.000000],accel_mss,speed_ms,0,0.000)
    |   movel(p[0.413680, -0.072103, -0.000100, 0.000000, -3.141593, 0.000000],accel_mss,speed_ms,0,0.000)
    |   movel(p[0.413748, -0.072229, -0.000100, 0.000000, -3.141593, 0.000000],accel_mss,speed_ms,0,0.000)
    |   movel(p[0.413823, -0.072360, -0.000100, 0.000000, -3.141593, 0.000000],accel_mss,speed_ms,0,0.000)
    |   movel(p[0.414031, -0.072638, -0.000100, 0.000000, -3.141593, 0.000000],accel_mss,speed_ms,0,0.000)
    |   movel(p[0.414287, -0.072962, -0.000100, 0.000000, -3.141593, 0.000000],accel_mss,speed_ms,0,0.000)
    |   movel(p[0.414573, -0.073305, -0.000100, 0.000000, -3.141593, 0.000000],accel_mss,speed_ms,0,0.000)
    |   movel(p[0.414852, -0.073640, -0.000100, 0.000000, -3.141593, 0.000000],accel_mss,speed_ms,0,0.000)
    |   movel(p[0.415087, -0.073945, -0.000100, 0.000000, -3.141593, 0.000000],accel_mss,speed_ms,0,0.000)
    |   movel(p[0.415274, -0.074206, -0.000100, 0.000000, -3.141593, 0.000000],accel_mss,speed_ms,0,0.000)
    |   movel(p[0.415322, -0.074364, -0.000100, 0.000000, -3.141593, 0.000000],accel_mss,speed_ms,0,0.000)
    |   movel(p[0.415411, -0.074490, -0.000100, 0.000000, -3.141593, 0.000000],accel_mss,speed_ms,0,0.000)
    |   movel(p[0.415532, -0.074634, -0.000100, 0.000000, -3.141593, 0.000000],accel_mss,speed_ms,0,0.000)
    |   movel(p[0.415676, -0.074779, -0.000100, 0.000000, -3.141593, 0.000000],accel_mss,speed_ms,0,0.000)
    |   movel(p[0.415819, -0.074926, -0.000100, 0.000000, 3.141593, 0.000000],accel_mss,speed_ms,0,0.000)
    |   movel(p[0.415940, -0.075078, -0.000100, 0.000000, 3.141593, 0.000000],accel_mss,speed_ms,0,0.000)
    |   movel(p[0.416027, -0.075214, -0.000100, 0.000000, -3.141593, 0.000000],accel_mss,speed_ms,0,0.000)
    |   movel(p[0.416077, -0.075393, -0.000100, 0.000000, -3.141593, 0.000000],accel_mss,speed_ms,0,0.000)
    |   movel(p[0.416183, -0.075549, -0.000100, 0.000000, -3.141593, 0.000000],accel_mss,speed_ms,0,0.000)
    |   movel(p[0.416328, -0.075726, -0.000100, 0.000000, -3.141593, 0.000000],accel_mss,speed_ms,0,0.000)
    |   movel(p[0.416501, -0.075904, -0.000100, 0.000000, -3.141593, 0.000000],accel_mss,speed_ms,0,0.000)
    |   movel(p[0.416673, -0.076079, -0.000100, 0.000000, -3.141593, 0.000000],accel_mss,speed_ms,0,0.000)
    |   movel(p[0.416818, -0.076249, -0.000100, 0.000000, -3.141593, 0.000000],accel_mss,speed_ms,0,0.000)
    |   movel(p[0.416927, -0.076397, -0.000100, 0.000000, -3.141593, 0.000000],accel_mss,speed_ms,0,0.000)
    |   movel(p[0.416982, -0.076565, -0.000100, 0.000000, -3.141593, 0.000000],accel_mss,speed_ms,0,0.000)
    |   movel(p[0.417259, -0.076915, -0.000100, 0.000000, -3.141593, 0.000000],accel_mss,speed_ms,0,0.000)
    |   movel(p[0.417598, -0.077322, -0.000100, 0.000000, -3.141593, 0.000000],accel_mss,speed_ms,0,0.000)
    |   movel(p[0.418001, -0.077779, -0.000100, 0.000000, -3.141593, 0.000000],accel_mss,speed_ms,0,0.000)
    |   movel(p[0.418403, -0.078235, -0.000100, 0.000000, 3.141593, 0.000000],accel_mss,speed_ms,0,0.000)
    |   movel(p[0.418742, -0.078642, -0.000100, 0.000000, -3.141593, 0.000000],accel_mss,speed_ms,0,0.000)
    |   movel(p[0.419020, -0.078992, -0.000100, 0.000000, -3.141593, 0.000000],accel_mss,speed_ms,0,0.000)
    |   movel(p[0.419078, -0.079161, -0.000100, 0.000000, -3.141593, 0.000000],accel_mss,speed_ms,0,0.000)
    |   movel(p[0.419227, -0.079350, -0.000100, 0.000000, -3.141593, 0.000000],accel_mss,speed_ms,0,0.000)
    |   movel(p[0.419421, -0.079569, -0.000100, 0.000000, -3.141593, 0.000000],accel_mss,speed_ms,0,0.000)
    |   movel(p[0.419651, -0.079804, -0.000100, 0.000000, -3.141593, 0.000000],accel_mss,speed_ms,0,0.000)
    |   movel(p[0.419880, -0.080040, -0.000100, 0.000000, -3.141593, 0.000000],accel_mss,speed_ms,0,0.000)
    |   movel(p[0.420074, -0.080265, -0.000100, 0.000000, -3.141593, 0.000000],accel_mss,speed_ms,0,0.000)
    |   movel(p[0.420221, -0.080460, -0.000100, 0.000000, -3.141593, 0.000000],accel_mss,speed_ms,0,0.000)
    |   movel(p[0.420284, -0.080649, -0.000100, 0.000000, -3.141593, 0.000000],accel_mss,speed_ms,0,0.000)
    |   movel(p[0.420475, -0.080886, -0.000100, 0.000000, -3.141593, 0.000000],accel_mss,speed_ms,0,0.000)
    |   movel(p[0.420722, -0.081163, -0.000100, 0.000000, 3.141593, 0.000000],accel_mss,speed_ms,0,0.000)
    |   movel(p[0.421015, -0.081460, -0.000100, 0.000000, -3.141593, 0.000000],accel_mss,speed_ms,0,0.000)
    |   movel(p[0.421315, -0.081763, -0.000100, 0.000000, -3.141593, 0.000000],accel_mss,speed_ms,0,0.000)
    |   movel(p[0.421584, -0.082061, -0.000100, 0.000000, -3.141593, 0.000000],accel_mss,speed_ms,0,0.000)
    |   movel(p[0.421798, -0.082320, -0.000100, 0.000000, -3.141593, 0.000000],accel_mss,speed_ms,0,0.000)
    |   movel(p[0.421879, -0.082461, -0.000100, 0.000000, -3.141593, 0.000000],accel_mss,speed_ms,0,0.000)
    |   movel(p[0.421981, -0.082630, -0.000100, 0.000000, -3.141593, 0.000000],accel_mss,speed_ms,0,0.000)
    |   movel(p[0.422577, -0.083302, -0.000100, 0.000000, 3.141593, 0.000000],accel_mss,speed_ms,0,0.000)
    |   movel(p[0.423289, -0.084084, -0.000100, 0.000000, 3.141593, 0.000000],accel_mss,speed_ms,0,0.000)
    |   movel(p[0.424115, -0.084962, -0.000100, 0.000000, -3.141593, 0.000000],accel_mss,speed_ms,0,0.000)
    |   movel(p[0.424933, -0.085831, -0.000100, 0.000000, -3.141593, 0.000000],accel_mss,speed_ms,0,0.000)
    |   movel(p[0.425623, -0.086582, -0.000100, 0.000000, -3.141593, 0.000000],accel_mss,speed_ms,0,0.000)
    |   movel(p[0.426219, -0.087244, -0.000100, 0.000000, -3.141593, 0.000000],accel_mss,speed_ms,0,0.000)
    |   movel(p[0.426334, -0.087530, -0.000100, 0.000000, -3.141593, 0.000000],accel_mss,speed_ms,0,0.000)
    |   movel(p[0.428539, -0.089740, -0.000100, 0.000000, -3.141593, 0.000000],accel_mss,speed_ms,0,blend_radius_m)
    |   movel(p[0.430749, -0.091945, -0.000100, 0.000000, -3.141593, 0.000000],accel_mss,speed_ms,0,blend_radius_m)
    |   movel(p[0.430951, -0.092029, -0.000100, 0.000000, -3.141593, 0.000000],accel_mss,speed_ms,0,0.000)
    |   movel(p[0.431561, -0.092514, -0.000100, 0.000000, -3.141593, 0.000000],accel_mss,speed_ms,0,0.000)
    |   movel(p[0.432159, -0.093046, -0.000100, 0.000000, -3.141593, 0.000000],accel_mss,speed_ms,0,0.000)
    |   movel(p[0.432844, -0.093679, -0.000100, 0.000000, -3.141593, 0.000000],accel_mss,speed_ms,0,0.000)
    |   movel(p[0.433530, -0.094311, -0.000100, 0.000000, -3.141593, 0.000000],accel_mss,speed_ms,0,0.000)
    |   movel(p[0.434130, -0.094844, -0.000100, 0.000000, -3.141593, 0.000000],accel_mss,speed_ms,0,0.000)
    |   movel(p[0.434654, -0.095294, -0.000100, 0.000000, -3.141593, 0.000000],accel_mss,speed_ms,0,0.000)
    |   movel(p[0.434748, -0.095329, -0.000100, 0.000000, -3.141593, 0.000000],accel_mss,speed_ms,0,0.000)
    |   movel(p[0.435041, -0.095527, -0.000100, 0.000000, -3.141593, 0.000000],accel_mss,speed_ms,0,0.000)
    |   movel(p[0.435287, -0.095745, -0.000100, 0.000000, -3.141593, 0.000000],accel_mss,speed_ms,0,0.000)
    |   movel(p[0.435551, -0.096004, -0.000100, 0.000000, -3.141593, 0.000000],accel_mss,speed_ms,0,0.000)
    |   movel(p[0.435816, -0.096262, -0.000100, 0.000000, 3.141593, 0.000000],accel_mss,speed_ms,0,0.000)
    |   movel(p[0.436066, -0.096481, -0.000100, 0.000000, -3.141593, 0.000000],accel_mss,speed_ms,0,0.000)
    |   movel(p[0.436280, -0.096648, -0.000100, 0.000000, -3.141593, 0.000000],accel_mss,speed_ms,0,0.000)
    |   movel(p[0.436472, -0.096712, -0.000100, 0.000000, -3.141593, 0.000000],accel_mss,speed_ms,0,0.000)
    |   movel(p[0.436728, -0.096921, -0.000100, 0.000000, -3.141593, 0.000000],accel_mss,speed_ms,0,0.000)
    |   movel(p[0.437027, -0.097188, -0.000100, 0.000000, -3.141593, 0.000000],accel_mss,speed_ms,0,0.000)
    |   movel(p[0.437351, -0.097504, -0.000100, 0.000000, -3.141593, 0.000000],accel_mss,speed_ms,0,0.000)
    |   movel(p[0.437676, -0.097820, -0.000100, 0.000000, -3.141593, 0.000000],accel_mss,speed_ms,0,0.000)
    |   movel(p[0.437979, -0.098087, -0.000100, 0.000000, -3.141593, 0.000000],accel_mss,speed_ms,0,0.000)
    |   movel(p[0.438239, -0.098293, -0.000100, 0.000000, -3.141593, 0.000000],accel_mss,speed_ms,0,0.000)
    |   movel(p[0.438346, -0.098329, -0.000100, 0.000000, -3.141593, 0.000000],accel_mss,speed_ms,0,0.000)
    |   movel(p[0.438649, -0.098454, -0.000100, 0.000000, -3.141593, 0.000000],accel_mss,speed_ms,0,0.000)
    |   movel(p[0.439504, -0.099301, -0.000100, 0.000000, -3.141593, 0.000000],accel_mss,speed_ms,0,0.000)
    |   movel(p[0.440358, -0.100148, -0.000100, 0.000000, -3.141593, 0.000000],accel_mss,speed_ms,0,0.000)
    |   movel(p[0.441212, -0.100995, -0.000100, 0.000000, -3.141593, 0.000000],accel_mss,speed_ms,0,0.000)
    |   movel(p[0.442065, -0.101843, -0.000100, 0.000000, -3.141593, 0.000000],accel_mss,speed_ms,0,0.000)
    |   movel(p[0.442918, -0.102692, -0.000100, 0.000000, -3.141593, 0.000000],accel_mss,speed_ms,0,0.000)
    |   movel(p[0.443771, -0.103540, -0.000100, 0.000000, -3.141593, 0.000000],accel_mss,speed_ms,0,0.000)
    |   movel(p[0.444624, -0.104389, -0.000100, 0.000000, -3.141593, 0.000000],accel_mss,speed_ms,0,0.000)
    |   movel(p[0.445476, -0.105239, -0.000100, 0.000000, -3.141593, 0.000000],accel_mss,speed_ms,0,0.000)
    |   movel(p[0.445601, -0.105540, -0.000100, 0.000000, -3.141593, 0.000000],accel_mss,speed_ms,0,0.000)
    |   movel(p[0.445683, -0.105768, -0.000100, 0.000000, -3.141593, 0.000000],accel_mss,speed_ms,0,0.000)
    |   movel(p[0.445774, -0.105911, -0.000100, 0.000000, -3.141593, 0.000000],accel_mss,speed_ms,0,0.000)
    |   movel(p[0.445882, -0.106044, -0.000100, 0.000000, -3.141593, 0.000000],accel_mss,speed_ms,0,0.000)
    |   movel(p[0.446105, -0.106332, -0.000100, 0.000000, -3.141593, 0.000000],accel_mss,speed_ms,0,0.000)
    |   movel(p[0.446412, -0.106820, -0.000100, 0.000000, -3.141593, 0.000000],accel_mss,speed_ms,0,0.000)
    |   movel(p[0.446786, -0.107470, -0.000100, 0.000000, -3.141593, 0.000000],accel_mss,speed_ms,0,0.000)
    |   movel(p[0.447237, -0.108304, -0.000100, 0.000000, -3.141593, 0.000000],accel_mss,speed_ms,0,0.000)
    |   movel(p[0.447445, -0.109017, -0.000100, 0.000000, -3.141593, 0.000000],accel_mss,speed_ms,0,0.000)
    |   movel(p[0.447489, -0.110283, -0.000100, 0.000000, -3.141593, 0.000000],accel_mss,speed_ms,0,0.001)
    |   movel(p[0.447412, -0.111560, -0.000100, 0.000000, -3.141593, 0.000000],accel_mss,speed_ms,0,0.001)
    |   movel(p[0.447188, -0.112354, -0.000100, 0.000000, -3.141593, 0.000000],accel_mss,speed_ms,0,0.000)
    |   movel(p[0.447050, -0.112649, -0.000100, 0.000000, -3.141593, 0.000000],accel_mss,speed_ms,0,0.000)
    |   movel(p[0.446861, -0.113053, -0.000100, 0.000000, -3.141593, 0.000000],accel_mss,speed_ms,0,0.000)
    |   movel(p[0.446658, -0.113489, -0.000100, 0.000000, -3.141593, 0.000000],accel_mss,speed_ms,0,0.000)
    |   movel(p[0.446470, -0.113891, -0.000100, 0.000000, -3.141593, 0.000000],accel_mss,speed_ms,0,0.000)
    |   movel(p[0.446293, -0.114251, -0.000100, 0.000000, -3.141593, 0.000000],accel_mss,speed_ms,0,0.000)
    |   movel(p[0.446121, -0.114554, -0.000100, 0.000000, -3.141593, 0.000000],accel_mss,speed_ms,0,0.000)
    |   movel(p[0.445967, -0.114790, -0.000100, 0.000000, -3.141593, 0.000000],accel_mss,speed_ms,0,0.000)
    |   movel(p[0.445839, -0.114844, -0.000100, 0.000000, -3.141593, 0.000000],accel_mss,speed_ms,0,0.000)
    |   movel(p[0.445761, -0.114952, -0.000100, 0.000000, -3.141593, 0.000000],accel_mss,speed_ms,0,0.000)
    |   movel(p[0.445726, -0.115127, -0.000100, 0.000000, -3.141593, 0.000000],accel_mss,speed_ms,0,0.000)
    |   movel(p[0.445640, -0.115272, -0.000100, 0.000000, -3.141593, 0.000000],accel_mss,speed_ms,0,0.000)
    |   movel(p[0.445519, -0.115429, -0.000100, 0.000000, -3.141593, 0.000000],accel_mss,speed_ms,0,0.000)
    |   movel(p[0.445376, -0.115579, -0.000100, 0.000000, -3.141593, 0.000000],accel_mss,speed_ms,0,0.000)
    |   movel(p[0.445232, -0.115726, -0.000100, 0.000000, -3.141593, 0.000000],accel_mss,speed_ms,0,0.000)
    |   movel(p[0.445111, -0.115878, -0.000100, 0.000000, -3.141593, 0.000000],accel_mss,speed_ms,0,0.000)
    |   movel(p[0.445024, -0.116015, -0.000100, 0.000000, -3.141593, 0.000000],accel_mss,speed_ms,0,0.000)
    |   movel(p[0.444888, -0.116375, -0.000100, 0.000000, -3.141593, 0.000000],accel_mss,speed_ms,0,0.000)
    |   movel(p[0.444389, -0.116832, -0.000100, 0.000000, -3.141593, 0.000000],accel_mss,speed_ms,0,0.000)
    |   movel(p[0.443628, -0.117416, -0.000100, 0.000000, -3.141593, 0.000000],accel_mss,speed_ms,0,0.000)
    |   movel(p[0.442526, -0.118170, -0.000100, 0.000000, -3.141593, 0.000000],accel_mss,speed_ms,0,0.001)
    |   movel(p[0.441762, -0.118587, -0.000100, 0.000000, -3.141593, 0.000000],accel_mss,speed_ms,0,0.000)
    |   movel(p[0.440786, -0.118965, -0.000100, 0.000000, -3.141593, 0.000000],accel_mss,speed_ms,0,0.000)
    |   movel(p[0.439738, -0.119258, -0.000100, 0.000000, -3.141593, 0.000000],accel_mss,speed_ms,0,0.000)
    |   movel(p[0.438751, -0.119422, -0.000100, 0.000000, -3.141593, 0.000000],accel_mss,speed_ms,0,0.000)
    |   movel(p[0.437377, -0.119409, -0.000100, 0.000000, -3.141593, 0.000000],accel_mss,speed_ms,0,0.001)
    |   movel(p[0.435645, -0.119097, -0.000100, 0.000000, -3.141593, 0.000000],accel_mss,speed_ms,0,0.001)
    |   movel(p[0.433882, -0.118576, -0.000100, 0.000000, -3.141593, 0.000000],accel_mss,speed_ms,0,0.001)
    |   movel(p[0.432395, -0.117912, -0.000100, 0.000000, -3.141593, 0.000000],accel_mss,speed_ms,0,0.001)
    |   movel(p[0.432001, -0.117700, -0.000100, 0.000000, -3.141593, 0.000000],accel_mss,speed_ms,0,0.000)
    |   movel(p[0.431620, -0.117499, -0.000100, 0.000000, -3.141593, 0.000000],accel_mss,speed_ms,0,0.000)
    |   movel(p[0.431294, -0.117331, -0.000100, 0.000000, -3.141593, 0.000000],accel_mss,speed_ms,0,0.000)
    |   movel(p[0.431119, -0.117248, -0.000100, 0.000000, -3.141593, 0.000000],accel_mss,speed_ms,0,0.000)
    |   movel(p[0.430988, -0.117178, -0.000100, 0.000000, -3.141593, 0.000000],accel_mss,speed_ms,0,0.000)
    |   movel(p[0.430845, -0.117080, -0.000100, 0.000000, -3.141593, 0.000000],accel_mss,speed_ms,0,0.000)
    |   movel(p[0.430712, -0.116972, -0.000100, 0.000000, -3.141593, 0.000000],accel_mss,speed_ms,0,0.000)
    |   movel(p[0.430614, -0.116870, -0.000100, 0.000000, -3.141593, 0.000000],accel_mss,speed_ms,0,0.000)
    |   movel(p[0.430526, -0.116777, -0.000100, 0.000000, -3.141593, 0.000000],accel_mss,speed_ms,0,0.000)
    |   movel(p[0.430426, -0.116700, -0.000100, 0.000000, -3.141593, 0.000000],accel_mss,speed_ms,0,0.000)
    |   movel(p[0.430331, -0.116645, -0.000100, 0.000000, -3.141593, 0.000000],accel_mss,speed_ms,0,0.000)
    |   movel(p[0.430159, -0.116599, -0.000100, 0.000000, -3.141593, 0.000000],accel_mss,speed_ms,0,0.000)
    |   movel(p[0.429892, -0.116409, -0.000100, 0.000000, -3.141593, 0.000000],accel_mss,speed_ms,0,0.000)
    |   movel(p[0.429578, -0.116166, -0.000100, 0.000000, -3.141593, 0.000000],accel_mss,speed_ms,0,0.000)
    |   movel(p[0.429237, -0.115879, -0.000100, 0.000000, -3.141593, 0.000000],accel_mss,speed_ms,0,0.000)
    |   movel(p[0.428897, -0.115592, -0.000100, 0.000000, -3.141593, 0.000000],accel_mss,speed_ms,0,0.000)
    |   movel(p[0.428590, -0.115349, -0.000100, 0.000000, -3.141593, 0.000000],accel_mss,speed_ms,0,0.000)
    |   movel(p[0.428327, -0.115155, -0.000100, 0.000000, -3.141593, 0.000000],accel_mss,speed_ms,0,0.000)
    |   movel(p[0.428164, -0.115099, -0.000100, 0.000000, -3.141593, 0.000000],accel_mss,speed_ms,0,0.000)
    |   movel(p[0.427871, -0.114843, -0.000100, 0.000000, -3.141593, 0.000000],accel_mss,speed_ms,0,0.000)
    |   movel(p[0.427530, -0.114528, -0.000100, 0.000000, -3.141593, 0.000000],accel_mss,speed_ms,0,0.000)
    |   movel(p[0.427151, -0.114154, -0.000100, 0.000000, -3.141593, 0.000000],accel_mss,speed_ms,0,0.000)
    |   movel(p[0.426769, -0.113780, -0.000100, 0.000000, -3.141593, 0.000000],accel_mss,speed_ms,0,0.000)
    |   movel(p[0.426424, -0.113465, -0.000100, 0.000000, -3.141593, 0.000000],accel_mss,speed_ms,0,0.000)
    |   movel(p[0.426127, -0.113213, -0.000100, 0.000000, -3.141593, 0.000000],accel_mss,speed_ms,0,0.000)
    |   movel(p[0.425803, -0.113086, -0.000100, 0.000000, -3.141593, 0.000000],accel_mss,speed_ms,0,0.000)
    |   movel(p[0.424867, -0.112167, -0.000100, 0.000000, -3.141593, 0.000000],accel_mss,speed_ms,0,0.001)
    |   movel(p[0.423944, -0.111234, -0.000100, 0.000000, -3.141593, 0.000000],accel_mss,speed_ms,0,0.001)
    |   movel(p[0.423851, -0.111004, -0.000100, 0.000000, -3.141593, 0.000000],accel_mss,speed_ms,0,0.000)
    |   movel(p[0.423814, -0.110905, -0.000100, 0.000000, -3.141593, 0.000000],accel_mss,speed_ms,0,0.000)
    |   movel(p[0.423520, -0.110564, -0.000100, 0.000000, -3.141593, 0.000000],accel_mss,speed_ms,0,0.000)
    |   movel(p[0.423157, -0.110169, -0.000100, 0.000000, -3.141593, 0.000000],accel_mss,speed_ms,0,0.000)
    |   movel(p[0.422726, -0.109729, -0.000100, 0.000000, -3.141593, 0.000000],accel_mss,speed_ms,0,0.000)
    |   movel(p[0.422294, -0.109291, -0.000100, 0.000000, -3.141593, 0.000000],accel_mss,speed_ms,0,0.000)
    |   movel(p[0.421931, -0.108901, -0.000100, 0.000000, -3.141593, 0.000000],accel_mss,speed_ms,0,0.000)
    |   movel(p[0.421632, -0.108564, -0.000100, 0.000000, -3.141593, 0.000000],accel_mss,speed_ms,0,0.000)
    |   movel(p[0.421569, -0.108392, -0.000100, 0.000000, -3.141593, 0.000000],accel_mss,speed_ms,0,0.000)
    |   movel(p[0.421226, -0.107978, -0.000100, 0.000000, -3.141593, 0.000000],accel_mss,speed_ms,0,0.000)
    |   movel(p[0.420814, -0.107500, -0.000100, 0.000000, -3.141593, 0.000000],accel_mss,speed_ms,0,0.000)
    |   movel(p[0.420326, -0.106958, -0.000100, 0.000000, -3.141593, 0.000000],accel_mss,speed_ms,0,0.000)
    |   movel(p[0.419837, -0.106416, -0.000100, 0.000000, -3.141593, 0.000000],accel_mss,speed_ms,0,0.000)
    |   movel(p[0.419425, -0.105937, -0.000100, 0.000000, -3.141593, 0.000000],accel_mss,speed_ms,0,0.000)
    |   movel(p[0.419083, -0.105522, -0.000100, 0.000000, -3.141593, 0.000000],accel_mss,speed_ms,0,0.000)
    |   movel(p[0.419021, -0.105347, -0.000100, 0.000000, -3.141593, 0.000000],accel_mss,speed_ms,0,0.000)
    |   movel(p[0.418830, -0.105116, -0.000100, 0.000000, -3.141593, 0.000000],accel_mss,speed_ms,0,0.000)
    |   movel(p[0.418588, -0.104847, -0.000100, 0.000000, -3.141593, 0.000000],accel_mss,speed_ms,0,0.000)
    |   movel(p[0.418301, -0.104554, -0.000100, 0.000000, -3.141593, 0.000000],accel_mss,speed_ms,0,0.000)
    |   movel(p[0.418013, -0.104259, -0.000100, 0.000000, -3.141593, 0.000000],accel_mss,speed_ms,0,0.000)
    |   movel(p[0.417771, -0.103986, -0.000100, 0.000000, -3.141593, 0.000000],accel_mss,speed_ms,0,0.000)
    |   movel(p[0.417583, -0.103751, -0.000100, 0.000000, -3.141593, 0.000000],accel_mss,speed_ms,0,0.000)
    |   movel(p[0.417450, -0.103413, -0.000100, 0.000000, -3.141593, 0.000000],accel_mss,speed_ms,0,0.000)
    |   movel(p[0.415920, -0.101877, -0.000100, 0.000000, -3.141593, 0.000000],accel_mss,speed_ms,0,0.001)
    |   movel(p[0.414465, -0.100446, -0.000100, 0.000000, -3.141593, 0.000000],accel_mss,speed_ms,0,0.001)
    |   movel(p[0.413936, -0.100051, -0.000100, 0.000000, -3.141593, 0.000000],accel_mss,speed_ms,0,0.000)
    |   movel(p[0.413221, -0.099672, -0.000100, 0.000000, -3.141593, 0.000000],accel_mss,speed_ms,0,0.000)
    |   movel(p[0.412641, -0.099421, -0.000100, 0.000000, -3.141593, 0.000000],accel_mss,speed_ms,0,0.000)
    |   movel(p[0.412151, -0.099276, -0.000100, 0.000000, -3.141593, 0.000000],accel_mss,speed_ms,0,0.000)
    |   movel(p[0.411718, -0.099229, -0.000100, 0.000000, -3.141593, 0.000000],accel_mss,speed_ms,0,0.000)
    |   movel(p[0.411481, -0.099240, -0.000100, 0.000000, -3.141593, 0.000000],accel_mss,speed_ms,0,0.000)
    |   movel(p[0.411267, -0.099274, -0.000100, 0.000000, -3.141593, 0.000000],accel_mss,speed_ms,0,0.000)
    |   movel(p[0.411097, -0.099322, -0.000100, 0.000000, -3.141593, 0.000000],accel_mss,speed_ms,0,0.000)
    |   movel(p[0.410980, -0.099435, -0.000100, 0.000000, -3.141593, 0.000000],accel_mss,speed_ms,0,0.000)
    |   movel(p[0.410874, -0.099487, -0.000100, 0.000000, 3.141593, 0.000000],accel_mss,speed_ms,0,0.000)
    |   movel(p[0.410516, -0.099485, -0.000100, 0.000000, -3.141593, 0.000000],accel_mss,speed_ms,0,0.000)
    |   movel(p[0.410036, -0.099861, -0.000100, 0.000000, -3.141593, 0.000000],accel_mss,speed_ms,0,0.000)
    |   movel(p[0.409556, -0.100414, -0.000100, 0.000000, -3.141593, 0.000000],accel_mss,speed_ms,0,0.000)
    |   movel(p[0.409204, -0.101029, -0.000100, 0.000000, -3.141593, 0.000000],accel_mss,speed_ms,0,0.000)
    |   movel(p[0.409154, -0.101131, -0.000100, 0.000000, -3.141593, 0.000000],accel_mss,speed_ms,0,0.000)
    |   movel(p[0.409082, -0.101254, -0.000100, 0.000000, -3.141593, 0.000000],accel_mss,speed_ms,0,0.000)
    |   movel(p[0.409002, -0.101376, -0.000100, 0.000000, -3.141593, 0.000000],accel_mss,speed_ms,0,0.000)
    |   movel(p[0.408926, -0.101479, -0.000100, 0.000000, -3.141593, 0.000000],accel_mss,speed_ms,0,0.000)
    |   movel(p[0.408746, -0.101805, -0.000100, 0.000000, -3.141593, 0.000000],accel_mss,speed_ms,0,0.000)
    |   movel(p[0.408453, -0.102681, -0.000100, 0.000000, -3.141593, 0.000000],accel_mss,speed_ms,0,0.000)
    |   movel(p[0.408144, -0.103729, -0.000100, 0.000000, -3.141593, 0.000000],accel_mss,speed_ms,0,0.000)
    |   movel(p[0.407856, -0.104854, -0.000100, 0.000000, -3.141593, 0.000000],accel_mss,speed_ms,0,0.000)
    |   movel(p[0.407677, -0.105985, -0.000100, 0.000000, -3.141593, 0.000000],accel_mss,speed_ms,0,0.000)
    |   movel(p[0.407572, -0.107775, -0.000100, 0.000000, -3.141593, 0.000000],accel_mss,speed_ms,0,0.001)
    |   movel(p[0.407541, -0.109552, -0.000100, 0.000000, -3.141593, 0.000000],accel_mss,speed_ms,0,0.001)
    |   movel(p[0.407643, -0.110554, -0.000100, 0.000000, -3.141593, 0.000000],accel_mss,speed_ms,0,0.000)
    |   movel(p[0.408221, -0.113193, -0.000100, 0.000000, -3.141593, 0.000000],accel_mss,speed_ms,0,blend_radius_m)
    |   movel(p[0.408843, -0.115588, -0.000100, 0.000000, -3.141593, 0.000000],accel_mss,speed_ms,0,0.001)
    |   movel(p[0.409447, -0.117551, -0.000100, 0.000000, -3.141593, 0.000000],accel_mss,speed_ms,0,0.001)
    |   movel(p[0.409937, -0.118654, -0.000100, 0.000000, -3.141593, 0.000000],accel_mss,speed_ms,0,0.000)
    |   movel(p[0.410024, -0.118812, -0.000100, 0.000000, -3.141593, 0.000000],accel_mss,speed_ms,0,0.000)
    |   movel(p[0.410154, -0.119055, -0.000100, 0.000000, -3.141593, 0.000000],accel_mss,speed_ms,0,0.000)
    |   movel(p[0.410299, -0.119330, -0.000100, 0.000000, -3.141593, 0.000000],accel_mss,speed_ms,0,0.000)
    |   movel(p[0.410437, -0.119599, -0.000100, 0.000000, -3.141593, 0.000000],accel_mss,speed_ms,0,0.000)
    |   movel(p[0.410579, -0.119864, -0.000100, 0.000000, -3.141593, 0.000000],accel_mss,speed_ms,0,0.000)
    |   movel(p[0.410730, -0.120129, -0.000100, 0.000000, -3.141593, 0.000000],accel_mss,speed_ms,0,0.000)
    |   movel(p[0.410871, -0.120358, -0.000100, 0.000000, -3.141593, 0.000000],accel_mss,speed_ms,0,0.000)
    |   movel(p[0.410971, -0.120499, -0.000100, 0.000000, -3.141593, 0.000000],accel_mss,speed_ms,0,0.000)
    |   movel(p[0.411340, -0.121059, -0.000100, 0.000000, -3.141593, 0.000000],accel_mss,speed_ms,0,0.000)
    |   movel(p[0.411420, -0.121490, -0.000100, 0.000000, -3.141593, 0.000000],accel_mss,speed_ms,0,0.000)
    |   movel(p[0.411242, -0.121918, -0.000100, 0.000000, -3.141593, 0.000000],accel_mss,speed_ms,0,0.000)
    |   movel(p[0.410732, -0.122479, -0.000100, 0.000000, -3.141593, 0.000000],accel_mss,speed_ms,0,0.000)
    |   movel(p[0.410403, -0.122767, -0.000100, 0.000000, -3.141593, 0.000000],accel_mss,speed_ms,0,0.000)
    |   movel(p[0.410154, -0.122911, -0.000100, 0.000000, -3.141593, 0.000000],accel_mss,speed_ms,0,0.000)
    |   movel(p[0.409878, -0.122974, -0.000100, 0.000000, -3.141593, 0.000000],accel_mss,speed_ms,0,0.000)
    |   movel(p[0.409460, -0.122982, -0.000100, 0.000000, -3.141593, 0.000000],accel_mss,speed_ms,0,0.000)
    |   movel(p[0.408862, -0.122909, -0.000100, 0.000000, -3.141593, 0.000000],accel_mss,speed_ms,0,0.000)
    |   movel(p[0.408270, -0.122727, -0.000100, 0.000000, -3.141593, 0.000000],accel_mss,speed_ms,0,0.000)
    |   movel(p[0.407600, -0.122406, -0.000100, 0.000000, -3.141593, 0.000000],accel_mss,speed_ms,0,0.000)
    |   movel(p[0.406751, -0.121895, -0.000100, 0.000000, -3.141593, 0.000000],accel_mss,speed_ms,0,0.000)
    |   movel(p[0.406396, -0.121672, -0.000100, 0.000000, -3.141593, 0.000000],accel_mss,speed_ms,0,0.000)
    |   movel(p[0.406014, -0.121439, -0.000100, 0.000000, -3.141593, 0.000000],accel_mss,speed_ms,0,0.000)
    |   movel(p[0.405659, -0.121228, -0.000100, 0.000000, -3.141593, 0.000000],accel_mss,speed_ms,0,0.000)
    |   movel(p[0.405401, -0.121082, -0.000100, 0.000000, -3.141593, 0.000000],accel_mss,speed_ms,0,0.000)
    |   movel(p[0.405177, -0.120952, -0.000100, 0.000000, -3.141593, 0.000000],accel_mss,speed_ms,0,0.000)
    |   movel(p[0.404939, -0.120798, -0.000100, 0.000000, -3.141593, 0.000000],accel_mss,speed_ms,0,0.000)
    |   movel(p[0.404722, -0.120642, -0.000100, 0.000000, -3.141593, 0.000000],accel_mss,speed_ms,0,0.000)
    |   movel(p[0.404566, -0.120513, -0.000100, 0.000000, -3.141593, 0.000000],accel_mss,speed_ms,0,0.000)
    |   movel(p[0.404434, -0.120404, -0.000100, 0.000000, -3.141593, 0.000000],accel_mss,speed_ms,0,0.000)
    |   movel(p[0.404293, -0.120312, -0.000100, 0.000000, -3.141593, 0.000000],accel_mss,speed_ms,0,0.000)
    |   movel(p[0.404162, -0.120248, -0.000100, 0.000000, -3.141593, 0.000000],accel_mss,speed_ms,0,0.000)
    |   movel(p[0.403775, -0.120108, -0.000100, 0.000000, -3.141593, 0.000000],accel_mss,speed_ms,0,0.000)
    |   movel(p[0.401939, -0.118280, -0.000100, 0.000000, -3.141593, 0.000000],accel_mss,speed_ms,0,blend_radius_m)
    |   movel(p[0.400191, -0.116509, -0.000100, 0.000000, -3.141593, 0.000000],accel_mss,speed_ms,0,0.001)
    |   movel(p[0.399848, -0.115999, -0.000100, 0.000000, -3.141593, 0.000000],accel_mss,speed_ms,0,0.000)
    |   movel(p[0.399769, -0.115835, -0.000100, 0.000000, -3.141593, 0.000000],accel_mss,speed_ms,0,0.000)
    |   movel(p[0.399655, -0.115623, -0.000100, 0.000000, -3.141593, 0.000000],accel_mss,speed_ms,0,0.000)
    |   movel(p[0.399527, -0.115401, -0.000100, 0.000000, -3.141593, 0.000000],accel_mss,speed_ms,0,0.000)
    |   movel(p[0.399404, -0.115204, -0.000100, 0.000000, -3.141593, 0.000000],accel_mss,speed_ms,0,0.000)
    |   movel(p[0.399027, -0.114557, -0.000100, 0.000000, -3.141593, 0.000000],accel_mss,speed_ms,0,0.000)
    |   movel(p[0.398553, -0.113611, -0.000100, 0.000000, -3.141593, 0.000000],accel_mss,speed_ms,0,0.000)
    |   movel(p[0.398111, -0.112646, -0.000100, 0.000000, -3.141593, 0.000000],accel_mss,speed_ms,0,0.000)
    |   movel(p[0.397839, -0.111937, -0.000100, 0.000000, -3.141593, 0.000000],accel_mss,speed_ms,0,0.000)
    |   movel(p[0.397436, -0.110518, -0.000100, 0.000000, -3.141593, 0.000000],accel_mss,speed_ms,0,0.001)
    |   movel(p[0.397159, -0.109075, -0.000100, 0.000000, -3.141593, 0.000000],accel_mss,speed_ms,0,0.001)
    |   movel(p[0.396974, -0.107380, -0.000100, 0.000000, -3.141593, 0.000000],accel_mss,speed_ms,0,0.001)
    |   movel(p[0.396848, -0.105154, -0.000100, 0.000000, -3.141593, 0.000000],accel_mss,speed_ms,0,0.001)
    |   movel(p[0.396786, -0.103797, -0.000100, 0.000000, -3.141593, 0.000000],accel_mss,speed_ms,0,0.001)
    |   movel(p[0.396710, -0.102449, -0.000100, 0.000000, -3.141593, 0.000000],accel_mss,speed_ms,0,0.001)
    |   movel(p[0.396631, -0.101278, -0.000100, 0.000000, -3.141593, 0.000000],accel_mss,speed_ms,0,0.000)
    |   movel(p[0.396564, -0.100579, -0.000100, 0.000000, 3.141593, 0.000000],accel_mss,speed_ms,0,0.000)
    |   movel(p[0.396206, -0.097793, -0.000100, 0.000000, -3.141593, 0.000000],accel_mss,speed_ms,0,blend_radius_m)
    |   movel(p[0.395875, -0.095761, -0.000100, 0.000000, -3.141593, 0.000000],accel_mss,speed_ms,0,0.001)
    |   movel(p[0.395501, -0.094053, -0.000100, 0.000000, -3.141593, 0.000000],accel_mss,speed_ms,0,0.001)
    |   movel(p[0.395016, -0.092329, -0.000100, 0.000000, -3.141593, 0.000000],accel_mss,speed_ms,0,0.001)
    |   movel(p[0.394606, -0.091152, -0.000100, 0.000000, -3.141593, 0.000000],accel_mss,speed_ms,0,0.000)
    |   movel(p[0.394110, -0.089969, -0.000100, 0.000000, -3.141593, 0.000000],accel_mss,speed_ms,0,0.001)
    |   movel(p[0.393619, -0.088954, -0.000100, 0.000000, -3.141593, 0.000000],accel_mss,speed_ms,0,0.000)
    |   movel(p[0.393301, -0.088558, -0.000100, 0.000000, -3.141593, 0.000000],accel_mss,speed_ms,0,0.000)
    |   movel(p[0.393224, -0.088482, -0.000100, 0.000000, -3.141593, 0.000000],accel_mss,speed_ms,0,0.000)
    |   movel(p[0.393159, -0.088390, -0.000100, 0.000000, -3.141593, 0.000000],accel_mss,speed_ms,0,0.000)
    |   movel(p[0.393115, -0.088297, -0.000100, 0.000000, -3.141593, 0.000000],accel_mss,speed_ms,0,0.000)
    |   movel(p[0.393065, -0.088114, -0.000100, 0.000000, -3.141593, 0.000000],accel_mss,speed_ms,0,0.000)
    |   movel(p[0.392847, -0.087845, -0.000100, 0.000000, -3.141593, 0.000000],accel_mss,speed_ms,0,0.000)
    |   movel(p[0.392569, -0.087531, -0.000100, 0.000000, 3.141593, 0.000000],accel_mss,speed_ms,0,0.000)
    |   movel(p[0.392238, -0.087191, -0.000100, 0.000000, -3.141593, 0.000000],accel_mss,speed_ms,0,0.000)
    |   movel(p[0.391782, -0.086758, -0.000100, 0.000000, -3.141593, 0.000000],accel_mss,speed_ms,0,0.000)
    |   movel(p[0.391482, -0.086528, -0.000100, 0.000000, -3.141593, 0.000000],accel_mss,speed_ms,0,0.000)
    |   movel(p[0.391250, -0.086426, -0.000100, 0.000000, -3.141593, 0.000000],accel_mss,speed_ms,0,0.000)
    |   movel(p[0.391038, -0.086426, -0.000100, 0.000000, -3.141593, 0.000000],accel_mss,speed_ms,0,0.000)
    |   movel(p[0.390909, -0.086470, -0.000100, 0.000000, -3.141593, 0.000000],accel_mss,speed_ms,0,0.000)
    |   movel(p[0.390800, -0.086531, -0.000100, 0.000000, -3.141593, 0.000000],accel_mss,speed_ms,0,0.000)
    |   movel(p[0.390724, -0.086598, -0.000100, 0.000000, -3.141593, 0.000000],accel_mss,speed_ms,0,0.000)
    |   movel(p[0.390668, -0.086754, -0.000100, 0.000000, -3.141593, 0.000000],accel_mss,speed_ms,0,0.000)
    |   movel(p[0.390392, -0.087098, -0.000100, 0.000000, -3.141593, 0.000000],accel_mss,speed_ms,0,0.000)
    |   movel(p[0.390053, -0.087498, -0.000100, 0.000000, -3.141593, 0.000000],accel_mss,speed_ms,0,0.000)
    |   movel(p[0.389651, -0.087946, -0.000100, 0.000000, -3.141593, 0.000000],accel_mss,speed_ms,0,0.000)
    |   movel(p[0.389248, -0.088391, -0.000100, 0.000000, -3.141593, 0.000000],accel_mss,speed_ms,0,0.000)
    |   movel(p[0.388909, -0.088784, -0.000100, 0.000000, -3.141593, 0.000000],accel_mss,speed_ms,0,0.000)
    |   movel(p[0.388627, -0.089124, -0.000100, 0.000000, -3.141593, 0.000000],accel_mss,speed_ms,0,0.000)
    |   movel(p[0.388582, -0.089272, -0.000100, 0.000000, -3.141593, 0.000000],accel_mss,speed_ms,0,0.000)
    |   movel(p[0.388468, -0.089476, -0.000100, 0.000000, 3.141593, 0.000000],accel_mss,speed_ms,0,0.000)
    |   movel(p[0.388323, -0.089717, -0.000100, 0.000000, -3.141593, 0.000000],accel_mss,speed_ms,0,0.000)
    |   movel(p[0.388151, -0.089981, -0.000100, 0.000000, -3.141593, 0.000000],accel_mss,speed_ms,0,0.000)
    |   movel(p[0.387978, -0.090245, -0.000100, 0.000000, 3.141593, 0.000000],accel_mss,speed_ms,0,0.000)
    |   movel(p[0.387833, -0.090488, -0.000100, 0.000000, -3.141593, 0.000000],accel_mss,speed_ms,0,0.000)
    |   movel(p[0.387720, -0.090694, -0.000100, 0.000000, -3.141593, 0.000000],accel_mss,speed_ms,0,0.000)
    |   movel(p[0.387621, -0.090968, -0.000100, 0.000000, -3.141593, 0.000000],accel_mss,speed_ms,0,0.000)
    |   movel(p[0.386912, -0.091690, -0.000100, 0.000000, -3.141593, 0.000000],accel_mss,speed_ms,0,0.000)
    |   movel(p[0.386189, -0.092400, -0.000100, 0.000000, -3.141593, 0.000000],accel_mss,speed_ms,0,0.000)
    |   movel(p[0.385993, -0.092479, -0.000100, 0.000000, -3.141593, 0.000000],accel_mss,speed_ms,0,0.000)
    |   movel(p[0.385810, -0.092552, -0.000100, 0.000000, -3.141593, 0.000000],accel_mss,speed_ms,0,0.000)
    |   movel(p[0.385690, -0.092633, -0.000100, 0.000000, 3.141593, 0.000000],accel_mss,speed_ms,0,0.000)
    |   movel(p[0.385574, -0.092728, -0.000100, 0.000000, -3.141593, 0.000000],accel_mss,speed_ms,0,0.000)
    |   movel(p[0.385332, -0.092923, -0.000100, 0.000000, -3.141593, 0.000000],accel_mss,speed_ms,0,0.000)
    |   movel(p[0.385048, -0.093110, -0.000100, 0.000000, -3.141593, 0.000000],accel_mss,speed_ms,0,0.000)
    |   movel(p[0.384652, -0.093331, -0.000100, 0.000000, 3.141593, 0.000000],accel_mss,speed_ms,0,0.000)
    |   movel(p[0.384026, -0.093652, -0.000100, 0.000000, -3.141593, 0.000000],accel_mss,speed_ms,0,0.000)
    |   movel(p[0.382206, -0.094461, -0.000100, 0.000000, -3.141593, 0.000000],accel_mss,speed_ms,0,0.001)
    |   movel(p[0.380511, -0.094997, -0.000100, 0.000000, -3.141593, 0.000000],accel_mss,speed_ms,0,0.001)
